LIN {X 0,Y 185.921,Z 403.304,A -85,B 0,C 180,E1 -22144.336,E2 -22144.336} C_VEL
LIN {X 0,Y 186.01,Z 403.316,A -85,B 0,C 180,E1 -22148.693,E2 -22148.693} C_VEL
LIN {X 0,Y 185.73,Z 403.33,A -85,B 0,C 180,E1 -22153.123,E2 -22153.123} C_VEL
LIN {X 0,Y 185.687,Z 403.347,A -85,B 0,C 180,E1 -22157.625,E2 -22157.625} C_VEL
LIN {X 0,Y 185.594,Z 403.365,A -85,B 0,C 180,E1 -22162.252,E2 -22162.252} C_VEL
LIN {X 0,Y 185.56,Z 403.358,A -85,B 0,C 180,E1 -22167.033,E2 -22167.033} C_VEL
LIN {X 0,Y 185.577,Z 403.368,A -85,B 0,C 180,E1 -22169.494,E2 -22169.494} C_VEL
LIN {X 0,Y 185.519,Z 403.376,A -85,B 0,C 180,E1 -22174.628,E2 -22174.628} C_VEL
LIN {X 0,Y 185.566,Z 403.36,A -85,B 0,C 180,E1 -22177.315,E2 -22177.315} C_VEL
LIN {X 0,Y 185.55,Z 403.372,A -85,B 0,C 180,E1 -22182.714,E2 -22182.714} C_VEL
LIN {X 0,Y 186.617,Z 406.323,A -85,B 0,C 180,E1 -22183.284,E2 -22183.284} C_VEL
LIN {X 0,Y 188.84,Z 408.797,A -85,B 0,C 180,E1 -22184.136,E2 -22184.136} C_VEL
LIN {X 0,Y 191.014,Z 412.188,A -85,B 0,C 180,E1 -22184.989,E2 -22184.989} C_VEL
LIN {X 0,Y 195.537,Z 418.863,A -85,B 0,C 180,E1 -22186.645,E2 -22186.645} C_VEL
LIN {X 0,Y 201.722,Z 428.495,A -85,B 0,C 180,E1 -22188.749,E2 -22188.749} C_VEL
LIN {X 0,Y 207.782,Z 439.318,A -85,B 0,C 180,E1 -22190.69,E2 -22190.69} C_VEL
LIN {X 0,Y 213.567,Z 452.7,A -85,B 0,C 180,E1 -22192.522,E2 -22192.522} C_VEL
LIN {X 0,Y 210.915,Z 504.609,A -85,B 0,C 180,E1 -22194.192,E2 -22194.192} C_VEL
LIN {X 0,Y 209.49,Z 518.077,A -85,B 0,C 180,E1 -22194.967,E2 -22194.967} C_VEL
LIN {X 0,Y 207.656,Z 530.461,A -85,B 0,C 180,E1 -22196.053,E2 -22196.053} C_VEL
LIN {X 0,Y 205.445,Z 541.745,A -85,B 0,C 180,E1 -22197.4,E2 -22197.4} C_VEL
LIN {X 0,Y 202.501,Z 553.363,A -85,B 0,C 180,E1 -22199.209,E2 -22199.209} C_VEL
LIN {X 0,Y 199.478,Z 563.795,A -85,B 0,C 180,E1 -22201.313,E2 -22201.313} C_VEL
LIN {X 0,Y 196.545,Z 573.207,A -85,B 0,C 180,E1 -22203.746,E2 -22203.746} C_VEL
LIN {X 0,Y 193.541,Z 581.541,A -85,B 0,C 180,E1 -22206.457,E2 -22206.457} C_VEL
LIN {X 0,Y 190.637,Z 588.935,A -85,B 0,C 180,E1 -22209.499,E2 -22209.499} C_VEL
LIN {X 0,Y 188.268,Z 594.864,A -85,B 0,C 180,E1 -22212.625,E2 -22212.625} C_VEL
LIN {X 0,Y 186.375,Z 599.545,A -85,B 0,C 180,E1 -22215.812,E2 -22215.812} C_VEL
LIN {X 0,Y 184.953,Z 603.125,A -85,B 0,C 180,E1 -22219.048,E2 -22219.048} C_VEL
LIN {X 0,Y 184.328,Z 604.97,A -85,B 0,C 180,E1 -22221.228,E2 -22221.228} C_VEL
LIN {X 0,Y 183.741,Z 606.644,A -85,B 0,C 180,E1 -22223.984,E2 -22223.984} C_VEL
LIN {X 0,Y 183.371,Z 607.945,A -85,B 0,C 180,E1 -22227.804,E2 -22227.804} C_VEL
LIN {X 0,Y 183.338,Z 608.171,A -85,B 0,C 180,E1 -22230,E2 -22230} C_VEL
LIN {X 0,Y 183.371,Z 607.978,A -85,B 0,C 180,E1 -22232.196,E2 -22232.196} C_VEL
LIN {X 0,Y 183.863,Z 606.429,A -85,B 0,C 180,E1 -22236.585,E2 -22236.585} C_VEL
LIN {X 0,Y 184.335,Z 605.076,A -85,B 0,C 180,E1 -22238.772,E2 -22238.772} C_VEL
LIN {X 0,Y 185.378,Z 602.216,A -85,B 0,C 180,E1 -22242.035,E2 -22242.035} C_VEL
LIN {X 0,Y 186.907,Z 598.332,A -85,B 0,C 180,E1 -22245.26,E2 -22245.26} C_VEL
LIN {X 0,Y 188.94,Z 593.319,A -85,B 0,C 180,E1 -22248.431,E2 -22248.431} C_VEL
LIN {X 0,Y 191.442,Z 587.001,A -85,B 0,C 180,E1 -22251.537,E2 -22251.537} C_VEL
LIN {X 0,Y 194.562,Z 579.089,A -85,B 0,C 180,E1 -22254.544,E2 -22254.544} C_VEL
LIN {X 0,Y 197.341,Z 570.784,A -85,B 0,C 180,E1 -22257.084,E2 -22257.084} C_VEL
LIN {X 0,Y 200.308,Z 561.19,A -85,B 0,C 180,E1 -22259.419,E2 -22259.419} C_VEL
LIN {X 0,Y 203.474,Z 550.096,A -85,B 0,C 180,E1 -22261.494,E2 -22261.494} C_VEL
LIN {X 0,Y 206.094,Z 539.217,A -85,B 0,C 180,E1 -22263.066,E2 -22263.066} C_VEL
LIN {X 0,Y 208.333,Z 527.192,A -85,B 0,C 180,E1 -22264.405,E2 -22264.405} C_VEL
LIN {X 0,Y 210.09,Z 514.712,A -85,B 0,C 180,E1 -22265.396,E2 -22265.396} C_VEL
LIN {X 0,Y 211.224,Z 502.268,A -85,B 0,C 180,E1 -22266.031,E2 -22266.031} C_VEL
LIN {X 0,Y 213.724,Z 452.937,A -85,B 0,C 180,E1 -22267.597,E2 -22267.597} C_VEL
LIN {X 0,Y 207.739,Z 439.055,A -85,B 0,C 180,E1 -22269.499,E2 -22269.499} C_VEL
LIN {X 0,Y 200.977,Z 427.208,A -85,B 0,C 180,E1 -22271.676,E2 -22271.676} C_VEL
LIN {X 0,Y 193.998,Z 416.477,A -85,B 0,C 180,E1 -22274.097,E2 -22274.097} C_VEL
LIN {X 0,Y 190.918,Z 412.068,A -85,B 0,C 180,E1 -22275.238,E2 -22275.238} C_VEL
LIN {X 0,Y 188.798,Z 408.673,A -85,B 0,C 180,E1 -22276.079,E2 -22276.079} C_VEL
LIN {X 0,Y 186.321,Z 405.856,A -85,B 0,C 180,E1 -22277.039,E2 -22277.039} C_VEL
LIN {X 0,Y 185.526,Z 403.347,A -85,B 0,C 180,E1 -22277.471,E2 -22277.471} C_VEL
LIN {X 0,Y 185.558,Z 403.363,A -85,B 0,C 180,E1 -22282.699,E2 -22282.699} C_VEL
LIN {X 0,Y 185.543,Z 403.368,A -85,B 0,C 180,E1 -22287.975,E2 -22287.975} C_VEL
LIN {X 0,Y 185.58,Z 403.361,A -85,B 0,C 180,E1 -22290.575,E2 -22290.575} C_VEL
LIN {X 0,Y 185.585,Z 403.361,A -85,B 0,C 180,E1 -22295.382,E2 -22295.382} C_VEL
LIN {X 0,Y 185.672,Z 403.349,A -85,B 0,C 180,E1 -22301.133,E2 -22301.133} C_VEL
LIN {X 0,Y 185.691,Z 403.351,A -85,B 0,C 180,E1 -22304.637,E2 -22304.637} C_VEL
LIN {X 0,Y 185.921,Z 403.311,A -85,B 0,C 180,E1 -22309.359,E2 -22309.359} C_VEL
LIN {X 0,Y 185.957,Z 403.316,A -85,B 0,C 180,E1 -22313.49,E2 -22313.49} C_VEL
LIN {X 0,Y 186.204,Z 403.289,A -85,B 0,C 180,E1 -22317.837,E2 -22317.837} C_VEL
LIN {X 0,Y 186.405,Z 403.263,A -85,B 0,C 180,E1 -22320,E2 -22320} C_VEL
LIN {X 0,Y 185.922,Z 403.322,A -85,B 0,C 180,E1 -22324.336,E2 -22324.336} C_VEL
LIN {X 0,Y 186.005,Z 403.299,A -85,B 0,C 180,E1 -22328.693,E2 -22328.693} C_VEL
LIN {X 0,Y 185.76,Z 403.336,A -85,B 0,C 180,E1 -22333.121,E2 -22333.121} C_VEL
LIN {X 0,Y 185.672,Z 403.347,A -85,B 0,C 180,E1 -22338.867,E2 -22338.867} C_VEL
LIN {X 0,Y 185.594,Z 403.367,A -85,B 0,C 180,E1 -22342.252,E2 -22342.252} C_VEL
LIN {X 0,Y 185.56,Z 403.371,A -85,B 0,C 180,E1 -22347.032,E2 -22347.032} C_VEL
LIN {X 0,Y 185.577,Z 403.367,A -85,B 0,C 180,E1 -22349.494,E2 -22349.494} C_VEL
LIN {X 0,Y 185.519,Z 403.368,A -85,B 0,C 180,E1 -22354.628,E2 -22354.628} C_VEL
LIN {X 0,Y 185.567,Z 403.437,A -85,B 0,C 180,E1 -22359.373,E2 -22359.373} C_VEL
LIN {X 0,Y 186.903,Z 408.111,A -85,B 0,C 180,E1 -22362.794,E2 -22362.794} C_VEL
LIN {X 0,Y 189.35,Z 412.41,A -85,B 0,C 180,E1 -22363.811,E2 -22363.811} C_VEL
LIN {X 0,Y 190.852,Z 414.784,A -85,B 0,C 180,E1 -22364.4,E2 -22364.4} C_VEL
LIN {X 0,Y 196.066,Z 423.736,A -85,B 0,C 180,E1 -22366.366,E2 -22366.366} C_VEL
LIN {X 0,Y 202.742,Z 436.785,A -85,B 0,C 180,E1 -22368.727,E2 -22368.727} C_VEL
LIN {X 0,Y 209.741,Z 452.959,A -85,B 0,C 180,E1 -22371.069,E2 -22371.069} C_VEL
LIN {X 0,Y 211.194,Z 456.662,A -85,B 0,C 180,E1 -22371.542,E2 -22371.542} C_VEL
LIN {X 0,Y 212.839,Z 470.861,A -85,B 0,C 180,E1 -22372.482,E2 -22372.482} C_VEL
LIN {X 0,Y 211.219,Z 504.612,A -85,B 0,C 180,E1 -22373.552,E2 -22373.552} C_VEL
LIN {X 0,Y 210.385,Z 510.464,A -85,B 0,C 180,E1 -22373.628,E2 -22373.628} C_VEL
LIN {X 0,Y 207.304,Z 519.917,A -85,B 0,C 180,E1 -22373.522,E2 -22373.522} C_VEL
LIN {X 0,Y 203.883,Z 529.234,A -85,B 0,C 180,E1 -22373.577,E2 -22373.577} C_VEL
LIN {X 0,Y 202.499,Z 534.867,A -85,B 0,C 180,E1 -22373.897,E2 -22373.897} C_VEL
LIN {X 0,Y 199.9,Z 547.969,A -85,B 0,C 180,E1 -22375.159,E2 -22375.159} C_VEL
LIN {X 0,Y 196.981,Z 559.755,A -85,B 0,C 180,E1 -22376.733,E2 -22376.733} C_VEL
LIN {X 0,Y 193.867,Z 570.352,A -85,B 0,C 180,E1 -22378.594,E2 -22378.594} C_VEL
LIN {X 0,Y 190.595,Z 580.039,A -85,B 0,C 180,E1 -22380.753,E2 -22380.753} C_VEL
LIN {X 0,Y 187.348,Z 588.873,A -85,B 0,C 180,E1 -22383.247,E2 -22383.247} C_VEL
LIN {X 0,Y 184.148,Z 597.424,A -85,B 0,C 180,E1 -22386.343,E2 -22386.343} C_VEL
LIN {X 0,Y 181.905,Z 603.374,A -85,B 0,C 180,E1 -22389.061,E2 -22389.061} C_VEL
LIN {X 0,Y 179.971,Z 608.236,A -85,B 0,C 180,E1 -22391.796,E2 -22391.796} C_VEL
LIN {X 0,Y 178.081,Z 612.962,A -85,B 0,C 180,E1 -22395.136,E2 -22395.136} C_VEL
LIN {X 0,Y 176.948,Z 616.585,A -85,B 0,C 180,E1 -22398.546,E2 -22398.546} C_VEL
LIN {X 0,Y 176.45,Z 618.455,A -85,B 0,C 180,E1 -22400.833,E2 -22400.833} C_VEL
LIN {X 0,Y 176.137,Z 619.86,A -85,B 0,C 180,E1 -22403.125,E2 -22403.125} C_VEL
LIN {X 0,Y 175.991,Z 621.264,A -85,B 0,C 180,E1 -22406.709,E2 -22406.709} C_VEL
LIN {X 0,Y 176.185,Z 621.701,A -85,B 0,C 180,E1 -22410,E2 -22410} C_VEL
LIN {X 0,Y 175.996,Z 621.246,A -85,B 0,C 180,E1 -22413.32,E2 -22413.32} C_VEL
LIN {X 0,Y 176.135,Z 619.831,A -85,B 0,C 180,E1 -22416.875,E2 -22416.875} C_VEL
LIN {X 0,Y 176.444,Z 618.412,A -85,B 0,C 180,E1 -22419.168,E2 -22419.168} C_VEL
LIN {X 0,Y 177.285,Z 615.445,A -85,B 0,C 180,E1 -22422.593,E2 -22422.593} C_VEL
LIN {X 0,Y 178.607,Z 611.438,A -85,B 0,C 180,E1 -22425.988,E2 -22425.988} C_VEL
LIN {X 0,Y 181.065,Z 605.294,A -85,B 0,C 180,E1 -22429.854,E2 -22429.854} C_VEL
LIN {X 0,Y 184.117,Z 597.764,A -85,B 0,C 180,E1 -22433.431,E2 -22433.431} C_VEL
LIN {X 0,Y 186.819,Z 590.279,A -85,B 0,C 180,E1 -22436.233,E2 -22436.233} C_VEL
LIN {X 0,Y 189.965,Z 581.763,A -85,B 0,C 180,E1 -22438.747,E2 -22438.747} C_VEL
LIN {X 0,Y 193.48,Z 571.246,A -85,B 0,C 180,E1 -22441.172,E2 -22441.172} C_VEL
LIN {X 0,Y 196.972,Z 559.412,A -85,B 0,C 180,E1 -22443.269,E2 -22443.269} C_VEL
LIN {X 0,Y 199.884,Z 547.485,A -85,B 0,C 180,E1 -22444.844,E2 -22444.844} C_VEL
LIN {X 0,Y 202.319,Z 535.072,A -85,B 0,C 180,E1 -22446.04,E2 -22446.04} C_VEL
LIN {X 0,Y 204.168,Z 522.069,A -85,B 0,C 180,E1 -22446.901,E2 -22446.901} C_VEL
LIN {X 0,Y 205.296,Z 506.698,A -85,B 0,C 180,E1 -22447.502,E2 -22447.502} C_VEL
LIN {X 0,Y 207.019,Z 471.198,A -85,B 0,C 180,E1 -22448.664,E2 -22448.664} C_VEL
LIN {X 0,Y 205.496,Z 458.664,A -85,B 0,C 180,E1 -22449.553,E2 -22449.553} C_VEL
LIN {X 0,Y 198.861,Z 442.643,A -85,B 0,C 180,E1 -22451.888,E2 -22451.888} C_VEL
LIN {X 0,Y 192.918,Z 430.579,A -85,B 0,C 180,E1 -22454.081,E2 -22454.081} C_VEL
LIN {X 0,Y 188.154,Z 422.026,A -85,B 0,C 180,E1 -22455.944,E2 -22455.944} C_VEL
LIN {X 0,Y 185.548,Z 417.623,A -85,B 0,C 180,E1 -22457.017,E2 -22457.017} C_VEL
LIN {X 0,Y 182.438,Z 412.577,A -85,B 0,C 180,E1 -22458.355,E2 -22458.355} C_VEL
LIN {X 0,Y 179.779,Z 408.407,A -85,B 0,C 180,E1 -22459.557,E2 -22459.557} C_VEL
LIN {X 0,Y 179.458,Z 407.656,A -85,B 0,C 180,E1 -22459.746,E2 -22459.746} C_VEL
LIN {X 0,Y 178.528,Z 404.239,A -85,B 0,C 180,E1 -22462.488,E2 -22462.488} C_VEL
LIN {X 0,Y 178.489,Z 404.24,A -85,B 0,C 180,E1 -22466.547,E2 -22466.547} C_VEL
LIN {X 0,Y 178.52,Z 404.239,A -85,B 0,C 180,E1 -22470.006,E2 -22470.006} C_VEL
LIN {X 0,Y 178.532,Z 404.238,A -85,B 0,C 180,E1 -22474.875,E2 -22474.875} C_VEL
LIN {X 0,Y 178.62,Z 404.229,A -85,B 0,C 180,E1 -22480.784,E2 -22480.784} C_VEL
LIN {X 0,Y 178.657,Z 404.231,A -85,B 0,C 180,E1 -22486.348,E2 -22486.348} C_VEL
LIN {X 0,Y 178.934,Z 404.179,A -85,B 0,C 180,E1 -22490.961,E2 -22490.961} C_VEL
LIN {X 0,Y 179.149,Z 404.148,A -85,B 0,C 180,E1 -22497.752,E2 -22497.752} C_VEL
LIN {X 0,Y 179.368,Z 404.14,A -85,B 0,C 180,E1 -22500,E2 -22500} C_VEL
LIN {X 0,Y 178.869,Z 404.181,A -85,B 0,C 180,E1 -22504.507,E2 -22504.507} C_VEL
LIN {X 0,Y 178.96,Z 404.192,A -85,B 0,C 180,E1 -22509.038,E2 -22509.038} C_VEL
LIN {X 0,Y 178.657,Z 404.214,A -85,B 0,C 180,E1 -22513.652,E2 -22513.652} C_VEL
LIN {X 0,Y 178.62,Z 404.215,A -85,B 0,C 180,E1 -22519.216,E2 -22519.216} C_VEL
LIN {X 0,Y 178.522,Z 404.232,A -85,B 0,C 180,E1 -22525.118,E2 -22525.118} C_VEL
LIN {X 0,Y 178.521,Z 404.242,A -85,B 0,C 180,E1 -22529.994,E2 -22529.994} C_VEL
LIN {X 0,Y 178.483,Z 404.253,A -85,B 0,C 180,E1 -22534.22,E2 -22534.22} C_VEL
LIN {X 0,Y 178.477,Z 404.249,A -85,B 0,C 180,E1 -22539.784,E2 -22539.784} C_VEL
LIN {X 0,Y 178.499,Z 404.253,A -85,B 0,C 180,E1 -22540.284,E2 -22540.284} C_VEL
LIN {X 0,Y 179.432,Z 406.939,A -85,B 0,C 180,E1 -22540.8,E2 -22540.8} C_VEL
LIN {X 0,Y 181.274,Z 409.049,A -85,B 0,C 180,E1 -22541.601,E2 -22541.601} C_VEL
LIN {X 0,Y 181.942,Z 409.687,A -85,B 0,C 180,E1 -22541.877,E2 -22541.877} C_VEL
LIN {X 0,Y 184.131,Z 413.133,A -85,B 0,C 180,E1 -22542.834,E2 -22542.834} C_VEL
LIN {X 0,Y 185.375,Z 414.712,A -85,B 0,C 180,E1 -22543.339,E2 -22543.339} C_VEL
LIN {X 0,Y 193.39,Z 426.657,A -85,B 0,C 180,E1 -22546.43,E2 -22546.43} C_VEL
LIN {X 0,Y 200.319,Z 438.22,A -85,B 0,C 180,E1 -22548.849,E2 -22548.849} C_VEL
LIN {X 0,Y 204.76,Z 447.222,A -85,B 0,C 180,E1 -22550.342,E2 -22550.342} C_VEL
LIN {X 0,Y 207.962,Z 454.895,A -85,B 0,C 180,E1 -22551.411,E2 -22551.411} C_VEL
LIN {X 0,Y 205.194,Z 505.053,A -85,B 0,C 180,E1 -22553.041,E2 -22553.041} C_VEL
LIN {X 0,Y 203.704,Z 518.479,A -85,B 0,C 180,E1 -22553.83,E2 -22553.83} C_VEL
LIN {X 0,Y 201.823,Z 530.735,A -85,B 0,C 180,E1 -22554.931,E2 -22554.931} C_VEL
LIN {X 0,Y 199.521,Z 542.016,A -85,B 0,C 180,E1 -22556.305,E2 -22556.305} C_VEL
LIN {X 0,Y 196.448,Z 553.634,A -85,B 0,C 180,E1 -22558.152,E2 -22558.152} C_VEL
LIN {X 0,Y 193.271,Z 564.066,A -85,B 0,C 180,E1 -22560.301,E2 -22560.301} C_VEL
LIN {X 0,Y 190.101,Z 573.75,A -85,B 0,C 180,E1 -22562.883,E2 -22562.883} C_VEL
LIN {X 0,Y 187.061,Z 581.81,A -85,B 0,C 180,E1 -22565.59,E2 -22565.59} C_VEL
LIN {X 0,Y 184.018,Z 589.204,A -85,B 0,C 180,E1 -22568.727,E2 -22568.727} C_VEL
LIN {X 0,Y 181.519,Z 595.132,A -85,B 0,C 180,E1 -22571.957,E2 -22571.957} C_VEL
LIN {X 0,Y 179.504,Z 599.814,A -85,B 0,C 180,E1 -22575.257,E2 -22575.257} C_VEL
LIN {X 0,Y 178.004,Z 603.393,A -85,B 0,C 180,E1 -22578.615,E2 -22578.615} C_VEL
LIN {X 0,Y 177.309,Z 605.238,A -85,B 0,C 180,E1 -22580.878,E2 -22580.878} C_VEL
LIN {X 0,Y 176.658,Z 607.052,A -85,B 0,C 180,E1 -22584.034,E2 -22584.034} C_VEL
LIN {X 0,Y 176.281,Z 608.213,A -85,B 0,C 180,E1 -22587.715,E2 -22587.715} C_VEL
LIN {X 0,Y 176.243,Z 608.438,A -85,B 0,C 180,E1 -22590,E2 -22590} C_VEL
LIN {X 0,Y 176.281,Z 608.245,A -85,B 0,C 180,E1 -22592.285,E2 -22592.285} C_VEL
LIN {X 0,Y 176.816,Z 606.696,A -85,B 0,C 180,E1 -22596.848,E2 -22596.848} C_VEL
LIN {X 0,Y 177.315,Z 605.343,A -85,B 0,C 180,E1 -22599.122,E2 -22599.122} C_VEL
LIN {X 0,Y 178.454,Z 602.481,A -85,B 0,C 180,E1 -22602.509,E2 -22602.509} C_VEL
LIN {X 0,Y 180.072,Z 598.598,A -85,B 0,C 180,E1 -22605.854,E2 -22605.854} C_VEL
LIN {X 0,Y 182.209,Z 593.585,A -85,B 0,C 180,E1 -22609.138,E2 -22609.138} C_VEL
LIN {X 0,Y 184.877,Z 587.266,A -85,B 0,C 180,E1 -22612.342,E2 -22612.342} C_VEL
LIN {X 0,Y 188.143,Z 579.353,A -85,B 0,C 180,E1 -22615.44,E2 -22615.44} C_VEL
LIN {X 0,Y 191.21,Z 570.575,A -85,B 0,C 180,E1 -22618.187,E2 -22618.187} C_VEL
LIN {X 0,Y 194.524,Z 560.352,A -85,B 0,C 180,E1 -22620.685,E2 -22620.685} C_VEL
LIN {X 0,Y 197.833,Z 548.937,A -85,B 0,C 180,E1 -22622.802,E2 -22622.802} C_VEL
LIN {X 0,Y 200.611,Z 537.717,A -85,B 0,C 180,E1 -22624.395,E2 -22624.395} C_VEL
LIN {X 0,Y 202.732,Z 526.313,A -85,B 0,C 180,E1 -22625.649,E2 -22625.649} C_VEL
LIN {X 0,Y 204.541,Z 513.346,A -85,B 0,C 180,E1 -22626.645,E2 -22626.645} C_VEL
LIN {X 0,Y 205.564,Z 501.19,A -85,B 0,C 180,E1 -22627.256,E2 -22627.256} C_VEL
LIN {X 0,Y 208.012,Z 454.901,A -85,B 0,C 180,E1 -22628.744,E2 -22628.744} C_VEL
LIN {X 0,Y 202.668,Z 442.523,A -85,B 0,C 180,E1 -22630.543,E2 -22630.543} C_VEL
LIN {X 0,Y 196.607,Z 431.784,A -85,B 0,C 180,E1 -22632.607,E2 -22632.607} C_VEL
LIN {X 0,Y 189.994,Z 421.47,A -85,B 0,C 180,E1 -22635.025,E2 -22635.025} C_VEL
LIN {X 0,Y 186.453,Z 416.413,A -85,B 0,C 180,E1 -22636.412,E2 -22636.412} C_VEL
LIN {X 0,Y 184.428,Z 413.419,A -85,B 0,C 180,E1 -22637.251,E2 -22637.251} C_VEL
LIN {X 0,Y 182.216,Z 410.251,A -85,B 0,C 180,E1 -22638.2,E2 -22638.2} C_VEL
LIN {X 0,Y 181.444,Z 409.171,A -85,B 0,C 180,E1 -22638.539,E2 -22638.539} C_VEL
LIN {X 0,Y 179.347,Z 406.852,A -85,B 0,C 180,E1 -22639.45,E2 -22639.45} C_VEL
LIN {X 0,Y 178.501,Z 404.246,A -85,B 0,C 180,E1 -22639.947,E2 -22639.947} C_VEL
LIN {X 0,Y 178.457,Z 404.252,A -85,B 0,C 180,E1 -22643.791,E2 -22643.791} C_VEL
LIN {X 0,Y 178.489,Z 404.242,A -85,B 0,C 180,E1 -22646.547,E2 -22646.547} C_VEL
LIN {X 0,Y 178.521,Z 404.244,A -85,B 0,C 180,E1 -22650.006,E2 -22650.006} C_VEL
LIN {X 0,Y 178.532,Z 404.244,A -85,B 0,C 180,E1 -22654.875,E2 -22654.875} C_VEL
LIN {X 0,Y 178.62,Z 404.23,A -85,B 0,C 180,E1 -22660.784,E2 -22660.784} C_VEL
LIN {X 0,Y 178.657,Z 404.23,A -85,B 0,C 180,E1 -22666.348,E2 -22666.348} C_VEL
LIN {X 0,Y 178.956,Z 404.189,A -85,B 0,C 180,E1 -22670.962,E2 -22670.962} C_VEL
LIN {X 0,Y 179.149,Z 404.166,A -85,B 0,C 180,E1 -22677.752,E2 -22677.752} C_VEL
LIN {X 0,Y 179.368,Z 404.138,A -85,B 0,C 180,E1 -22680,E2 -22680} C_VEL
LIN {X 0,Y 178.87,Z 404.201,A -85,B 0,C 180,E1 -22684.507,E2 -22684.507} C_VEL
LIN {X 0,Y 178.934,Z 404.18,A -85,B 0,C 180,E1 -22689.039,E2 -22689.039} C_VEL
LIN {X 0,Y 178.678,Z 404.215,A -85,B 0,C 180,E1 -22693.651,E2 -22693.651} C_VEL
LIN {X 0,Y 178.62,Z 404.223,A -85,B 0,C 180,E1 -22699.216,E2 -22699.216} C_VEL
LIN {X 0,Y 178.522,Z 404.238,A -85,B 0,C 180,E1 -22705.118,E2 -22705.118} C_VEL
LIN {X 0,Y 178.52,Z 404.245,A -85,B 0,C 180,E1 -22709.994,E2 -22709.994} C_VEL
LIN {X 0,Y 178.483,Z 404.241,A -85,B 0,C 180,E1 -22714.22,E2 -22714.22} C_VEL
LIN {X 0,Y 178.544,Z 404.366,A -85,B 0,C 180,E1 -22717.515,E2 -22717.515} C_VEL
LIN {X 0,Y 179.463,Z 407.711,A -85,B 0,C 180,E1 -22720.161,E2 -22720.161} C_VEL
LIN {X 0,Y 182.34,Z 412.457,A -85,B 0,C 180,E1 -22721.488,E2 -22721.488} C_VEL
LIN {X 0,Y 184.139,Z 415.339,A -85,B 0,C 180,E1 -22722.275,E2 -22722.275} C_VEL
LIN {X 0,Y 186.975,Z 419.928,A -85,B 0,C 180,E1 -22723.465,E2 -22723.465} C_VEL
LIN {X 0,Y 192.107,Z 429.035,A -85,B 0,C 180,E1 -22725.511,E2 -22725.511} C_VEL
LIN {X 0,Y 197.957,Z 440.605,A -85,B 0,C 180,E1 -22727.694,E2 -22727.694} C_VEL
LIN {X 0,Y 204.803,Z 456.726,A -85,B 0,C 180,E1 -22730.123,E2 -22730.123} C_VEL
LIN {X 0,Y 205.871,Z 459.872,A -85,B 0,C 180,E1 -22730.507,E2 -22730.507} C_VEL
LIN {X 0,Y 207.17,Z 472.203,A -85,B 0,C 180,E1 -22731.337,E2 -22731.337} C_VEL
LIN {X 0,Y 204.731,Z 518.229,A -85,B 0,C 180,E1 -22732.882,E2 -22732.882} C_VEL
LIN {X 0,Y 203.028,Z 531.674,A -85,B 0,C 180,E1 -22733.656,E2 -22733.656} C_VEL
LIN {X 0,Y 202.499,Z 534.867,A -85,B 0,C 180,E1 -22733.897,E2 -22733.897} C_VEL
LIN {X 0,Y 200.968,Z 540.521,A -85,B 0,C 180,E1 -22734.284,E2 -22734.284} C_VEL
LIN {X 0,Y 196.735,Z 549.398,A -85,B 0,C 180,E1 -22734.769,E2 -22734.769} C_VEL
LIN {X 0,Y 192.146,Z 557.81,A -85,B 0,C 180,E1 -22735.426,E2 -22735.426} C_VEL
LIN {X 0,Y 190.103,Z 562.779,A -85,B 0,C 180,E1 -22736.1,E2 -22736.1} C_VEL
LIN {X 0,Y 186.67,Z 573.565,A -85,B 0,C 180,E1 -22738.192,E2 -22738.192} C_VEL
LIN {X 0,Y 183.027,Z 583.515,A -85,B 0,C 180,E1 -22740.688,E2 -22740.688} C_VEL
LIN {X 0,Y 179.796,Z 591.68,A -85,B 0,C 180,E1 -22743.288,E2 -22743.288} C_VEL
LIN {X 0,Y 176.715,Z 599.71,A -85,B 0,C 180,E1 -22746.566,E2 -22746.566} C_VEL
LIN {X 0,Y 173.989,Z 606.143,A -85,B 0,C 180,E1 -22749.92,E2 -22749.92} C_VEL
LIN {X 0,Y 171.777,Z 611.256,A -85,B 0,C 180,E1 -22753.358,E2 -22753.358} C_VEL
LIN {X 0,Y 170.313,Z 615.238,A -85,B 0,C 180,E1 -22756.882,E2 -22756.882} C_VEL
LIN {X 0,Y 169.406,Z 618.187,A -85,B 0,C 180,E1 -22760.448,E2 -22760.448} C_VEL
LIN {X 0,Y 169.071,Z 619.592,A -85,B 0,C 180,E1 -22762.836,E2 -22762.836} C_VEL
LIN {X 0,Y 168.899,Z 621.092,A -85,B 0,C 180,E1 -22767.028,E2 -22767.028} C_VEL
LIN {X 0,Y 169.089,Z 621.434,A -85,B 0,C 180,E1 -22770,E2 -22770} C_VEL
LIN {X 0,Y 168.93,Z 621.04,A -85,B 0,C 180,E1 -22773.163,E2 -22773.163} C_VEL
LIN {X 0,Y 169.068,Z 619.562,A -85,B 0,C 180,E1 -22777.164,E2 -22777.164} C_VEL
LIN {X 0,Y 169.401,Z 618.143,A -85,B 0,C 180,E1 -22779.552,E2 -22779.552} C_VEL
LIN {X 0,Y 170.311,Z 615.175,A -85,B 0,C 180,E1 -22783.118,E2 -22783.118} C_VEL
LIN {X 0,Y 171.774,Z 611.169,A -85,B 0,C 180,E1 -22786.642,E2 -22786.642} C_VEL
LIN {X 0,Y 174.355,Z 605.024,A -85,B 0,C 180,E1 -22790.652,E2 -22790.652} C_VEL
LIN {X 0,Y 177.339,Z 598.098,A -85,B 0,C 180,E1 -22794.079,E2 -22794.079} C_VEL
LIN {X 0,Y 180.452,Z 590.008,A -85,B 0,C 180,E1 -22797.233,E2 -22797.233} C_VEL
LIN {X 0,Y 183.76,Z 581.492,A -85,B 0,C 180,E1 -22799.814,E2 -22799.814} C_VEL
LIN {X 0,Y 187.445,Z 570.976,A -85,B 0,C 180,E1 -22802.294,E2 -22802.294} C_VEL
LIN {X 0,Y 190.655,Z 560.572,A -85,B 0,C 180,E1 -22804.204,E2 -22804.204} C_VEL
LIN {X 0,Y 193.66,Z 549.159,A -85,B 0,C 180,E1 -22805.815,E2 -22805.815} C_VEL
LIN {X 0,Y 196.154,Z 537.4,A -85,B 0,C 180,E1 -22807.039,E2 -22807.039} C_VEL
LIN {X 0,Y 198.273,Z 523.822,A -85,B 0,C 180,E1 -22808.016,E2 -22808.016} C_VEL
LIN {X 0,Y 199.49,Z 510.457,A -85,B 0,C 180,E1 -22808.611,E2 -22808.611} C_VEL
LIN {X 0,Y 201.467,Z 472.332,A -85,B 0,C 180,E1 -22809.874,E2 -22809.874} C_VEL
LIN {X 0,Y 200.186,Z 461.38,A -85,B 0,C 180,E1 -22810.682,E2 -22810.682} C_VEL
LIN {X 0,Y 193.754,Z 445.675,A -85,B 0,C 180,E1 -22813.093,E2 -22813.093} C_VEL
LIN {X 0,Y 187.871,Z 433.538,A -85,B 0,C 180,E1 -22815.418,E2 -22815.418} C_VEL
LIN {X 0,Y 181.729,Z 422.646,A -85,B 0,C 180,E1 -22818.022,E2 -22818.022} C_VEL
LIN {X 0,Y 178.684,Z 417.711,A -85,B 0,C 180,E1 -22819.403,E2 -22819.403} C_VEL
LIN {X 0,Y 175.209,Z 412.284,A -85,B 0,C 180,E1 -22821.077,E2 -22821.077} C_VEL
LIN {X 0,Y 172.553,Z 408.312,A -85,B 0,C 180,E1 -22822.434,E2 -22822.434} C_VEL
LIN {X 0,Y 172.071,Z 407.183,A -85,B 0,C 180,E1 -22822.771,E2 -22822.771} C_VEL
LIN {X 0,Y 171.426,Z 405.132,A -85,B 0,C 180,E1 -22824.794,E2 -22824.794} C_VEL
LIN {X 0,Y 171.456,Z 405.124,A -85,B 0,C 180,E1 -22829.404,E2 -22829.404} C_VEL
LIN {X 0,Y 171.467,Z 405.123,A -85,B 0,C 180,E1 -22834.383,E2 -22834.383} C_VEL
LIN {X 0,Y 171.576,Z 405.105,A -85,B 0,C 180,E1 -22840.871,E2 -22840.871} C_VEL
LIN {X 0,Y 171.574,Z 405.113,A -85,B 0,C 180,E1 -22845.773,E2 -22845.773} C_VEL
LIN {X 0,Y 171.869,Z 405.056,A -85,B 0,C 180,E1 -22850.586,E2 -22850.586} C_VEL
LIN {X 0,Y 171.817,Z 405.07,A -85,B 0,C 180,E1 -22855.308,E2 -22855.308} C_VEL
LIN {X 0,Y 172.331,Z 405.017,A -85,B 0,C 180,E1 -22860,E2 -22860} C_VEL
LIN {X 0,Y 171.818,Z 405.059,A -85,B 0,C 180,E1 -22864.693,E2 -22864.693} C_VEL
LIN {X 0,Y 171.887,Z 405.072,A -85,B 0,C 180,E1 -22869.413,E2 -22869.413} C_VEL
LIN {X 0,Y 171.574,Z 405.102,A -85,B 0,C 180,E1 -22874.228,E2 -22874.228} C_VEL
LIN {X 0,Y 171.541,Z 405.096,A -85,B 0,C 180,E1 -22879.562,E2 -22879.562} C_VEL
LIN {X 0,Y 171.46,Z 405.109,A -85,B 0,C 180,E1 -22885.612,E2 -22885.612} C_VEL
LIN {X 0,Y 171.439,Z 405.119,A -85,B 0,C 180,E1 -22890.587,E2 -22890.587} C_VEL
LIN {X 0,Y 171.433,Z 405.119,A -85,B 0,C 180,E1 -22896.473,E2 -22896.473} C_VEL
LIN {X 0,Y 171.42,Z 405.121,A -85,B 0,C 180,E1 -22897.394,E2 -22897.394} C_VEL
LIN {X 0,Y 172.504,Z 408.032,A -85,B 0,C 180,E1 -22898.101,E2 -22898.101} C_VEL
LIN {X 0,Y 174.511,Z 410.147,A -85,B 0,C 180,E1 -22899.078,E2 -22899.078} C_VEL
LIN {X 0,Y 175.23,Z 410.924,A -85,B 0,C 180,E1 -22899.419,E2 -22899.419} C_VEL
LIN {X 0,Y 177.341,Z 414.18,A -85,B 0,C 180,E1 -22900.451,E2 -22900.451} C_VEL
LIN {X 0,Y 178.765,Z 415.871,A -85,B 0,C 180,E1 -22901.09,E2 -22901.09} C_VEL
LIN {X 0,Y 182.731,Z 421.675,A -85,B 0,C 180,E1 -22902.842,E2 -22902.842} C_VEL
LIN {X 0,Y 189.016,Z 431.038,A -85,B 0,C 180,E1 -22905.373,E2 -22905.373} C_VEL
LIN {X 0,Y 195.768,Z 442.518,A -85,B 0,C 180,E1 -22907.872,E2 -22907.872} C_VEL
LIN {X 0,Y 200.089,Z 451.464,A -85,B 0,C 180,E1 -22909.41,E2 -22909.41} C_VEL
LIN {X 0,Y 202.342,Z 456.987,A -85,B 0,C 180,E1 -22910.211,E2 -22910.211} C_VEL
LIN {X 0,Y 199.529,Z 505.635,A -85,B 0,C 180,E1 -22911.828,E2 -22911.828} C_VEL
LIN {X 0,Y 198.009,Z 518.889,A -85,B 0,C 180,E1 -22912.63,E2 -22912.63} C_VEL
LIN {X 0,Y 196.065,Z 531.009,A -85,B 0,C 180,E1 -22913.741,E2 -22913.741} C_VEL
LIN {X 0,Y 193.669,Z 542.288,A -85,B 0,C 180,E1 -22915.143,E2 -22915.143} C_VEL
LIN {X 0,Y 190.466,Z 553.905,A -85,B 0,C 180,E1 -22917.027,E2 -22917.027} C_VEL
LIN {X 0,Y 187.134,Z 564.337,A -85,B 0,C 180,E1 -22919.224,E2 -22919.224} C_VEL
LIN {X 0,Y 184.207,Z 572.891,A -85,B 0,C 180,E1 -22921.531,E2 -22921.531} C_VEL
LIN {X 0,Y 181.213,Z 580.697,A -85,B 0,C 180,E1 -22924.132,E2 -22924.132} C_VEL
LIN {X 0,Y 177.887,Z 588.365,A -85,B 0,C 180,E1 -22927.344,E2 -22927.344} C_VEL
LIN {X 0,Y 174.774,Z 595.401,A -85,B 0,C 180,E1 -22931.235,E2 -22931.235} C_VEL
LIN {X 0,Y 172.659,Z 600.082,A -85,B 0,C 180,E1 -22934.658,E2 -22934.658} C_VEL
LIN {X 0,Y 171.053,Z 603.66,A -85,B 0,C 180,E1 -22938.145,E2 -22938.145} C_VEL
LIN {X 0,Y 170.292,Z 605.506,A -85,B 0,C 180,E1 -22940.498,E2 -22940.498} C_VEL
LIN {X 0,Y 169.505,Z 607.564,A -85,B 0,C 180,E1 -22944.32,E2 -22944.32} C_VEL
LIN {X 0,Y 169.194,Z 608.48,A -85,B 0,C 180,E1 -22947.619,E2 -22947.619} C_VEL
LIN {X 0,Y 169.151,Z 608.705,A -85,B 0,C 180,E1 -22950,E2 -22950} C_VEL
LIN {X 0,Y 169.194,Z 608.511,A -85,B 0,C 180,E1 -22952.381,E2 -22952.381} C_VEL
LIN {X 0,Y 169.783,Z 606.962,A -85,B 0,C 180,E1 -22957.133,E2 -22957.133} C_VEL
LIN {X 0,Y 170.298,Z 605.61,A -85,B 0,C 180,E1 -22959.501,E2 -22959.501} C_VEL
LIN {X 0,Y 171.525,Z 602.748,A -85,B 0,C 180,E1 -22963.023,E2 -22963.023} C_VEL
LIN {X 0,Y 173.263,Z 598.864,A -85,B 0,C 180,E1 -22966.495,E2 -22966.495} C_VEL
LIN {X 0,Y 175.513,Z 593.851,A -85,B 0,C 180,E1 -22969.898,E2 -22969.898} C_VEL
LIN {X 0,Y 178.337,Z 587.531,A -85,B 0,C 180,E1 -22973.208,E2 -22973.208} C_VEL
LIN {X 0,Y 181.767,Z 579.617,A -85,B 0,C 180,E1 -22976.4,E2 -22976.4} C_VEL
LIN {X 0,Y 184.887,Z 571.093,A -85,B 0,C 180,E1 -22979.153,E2 -22979.153} C_VEL
LIN {X 0,Y 188.094,Z 561.716,A -85,B 0,C 180,E1 -22981.54,E2 -22981.54} C_VEL
LIN {X 0,Y 191.544,Z 550.619,A -85,B 0,C 180,E1 -22983.707,E2 -22983.707} C_VEL
LIN {X 0,Y 194.385,Z 539.738,A -85,B 0,C 180,E1 -22985.343,E2 -22985.343} C_VEL
LIN {X 0,Y 196.819,Z 527.71,A -85,B 0,C 180,E1 -22986.733,E2 -22986.733} C_VEL
LIN {X 0,Y 198.694,Z 515.395,A -85,B 0,C 180,E1 -22987.751,E2 -22987.751} C_VEL
LIN {X 0,Y 199.952,Z 501.977,A -85,B 0,C 180,E1 -22988.46,E2 -22988.46} C_VEL
LIN {X 0,Y 202.429,Z 457.041,A -85,B 0,C 180,E1 -22989.938,E2 -22989.938} C_VEL
LIN {X 0,Y 197.576,Z 445.864,A -85,B 0,C 180,E1 -22991.669,E2 -22991.669} C_VEL
LIN {X 0,Y 190.944,Z 434.057,A -85,B 0,C 180,E1 -22994.087,E2 -22994.087} C_VEL
LIN {X 0,Y 183.585,Z 422.785,A -85,B 0,C 180,E1 -22997.008,E2 -22997.008} C_VEL
LIN {X 0,Y 180.713,Z 418.712,A -85,B 0,C 180,E1 -22998.241,E2 -22998.241} C_VEL
LIN {X 0,Y 177.941,Z 414.782,A -85,B 0,C 180,E1 -22999.499,E2 -22999.499} C_VEL
LIN {X 0,Y 175.597,Z 411.667,A -85,B 0,C 180,E1 -23000.608,E2 -23000.608} C_VEL
LIN {X 0,Y 174.824,Z 410.346,A -85,B 0,C 180,E1 -23001.005,E2 -23001.005} C_VEL
LIN {X 0,Y 172.683,Z 408.34,A -85,B 0,C 180,E1 -23002.032,E2 -23002.032} C_VEL
LIN {X 0,Y 171.603,Z 406.109,A -85,B 0,C 180,E1 -23002.652,E2 -23002.652} C_VEL
LIN {X 0,Y 171.407,Z 405.125,A -85,B 0,C 180,E1 -23002.833,E2 -23002.833} C_VEL
LIN {X 0,Y 171.426,Z 405.124,A -85,B 0,C 180,E1 -23007.794,E2 -23007.794} C_VEL
LIN {X 0,Y 171.447,Z 405.12,A -85,B 0,C 180,E1 -23010.534,E2 -23010.534} C_VEL
LIN {X 0,Y 171.455,Z 405.117,A -85,B 0,C 180,E1 -23015.801,E2 -23015.801} C_VEL
LIN {X 0,Y 171.576,Z 405.106,A -85,B 0,C 180,E1 -23020.871,E2 -23020.871} C_VEL
LIN {X 0,Y 171.575,Z 405.113,A -85,B 0,C 180,E1 -23025.772,E2 -23025.772} C_VEL
LIN {X 0,Y 171.885,Z 405.066,A -85,B 0,C 180,E1 -23030.587,E2 -23030.587} C_VEL
LIN {X 0,Y 171.817,Z 405.065,A -85,B 0,C 180,E1 -23035.307,E2 -23035.307} C_VEL
LIN {X 0,Y 172.331,Z 405.014,A -85,B 0,C 180,E1 -23040,E2 -23040} C_VEL
LIN {X 0,Y 171.819,Z 405.08,A -85,B 0,C 180,E1 -23044.692,E2 -23044.692} C_VEL
LIN {X 0,Y 171.87,Z 405.062,A -85,B 0,C 180,E1 -23049.414,E2 -23049.414} C_VEL
LIN {X 0,Y 171.59,Z 405.095,A -85,B 0,C 180,E1 -23054.226,E2 -23054.226} C_VEL
LIN {X 0,Y 171.541,Z 405.104,A -85,B 0,C 180,E1 -23059.562,E2 -23059.562} C_VEL
LIN {X 0,Y 171.46,Z 405.119,A -85,B 0,C 180,E1 -23065.612,E2 -23065.612} C_VEL
LIN {X 0,Y 171.439,Z 405.126,A -85,B 0,C 180,E1 -23070.587,E2 -23070.587} C_VEL
LIN {X 0,Y 171.435,Z 405.284,A -85,B 0,C 180,E1 -23075.384,E2 -23075.384} C_VEL
LIN {X 0,Y 172.177,Z 407.394,A -85,B 0,C 180,E1 -23077.202,E2 -23077.202} C_VEL
LIN {X 0,Y 174.263,Z 411.108,A -85,B 0,C 180,E1 -23078.329,E2 -23078.329} C_VEL
LIN {X 0,Y 176.379,Z 413.97,A -85,B 0,C 180,E1 -23079.363,E2 -23079.363} C_VEL
LIN {X 0,Y 180.289,Z 420.239,A -85,B 0,C 180,E1 -23081.213,E2 -23081.213} C_VEL
LIN {X 0,Y 185.2,Z 428.558,A -85,B 0,C 180,E1 -23083.365,E2 -23083.365} C_VEL
LIN {X 0,Y 192.242,Z 442.247,A -85,B 0,C 180,E1 -23086.221,E2 -23086.221} C_VEL
LIN {X 0,Y 198.528,Z 456.956,A -85,B 0,C 180,E1 -23088.617,E2 -23088.617} C_VEL
LIN {X 0,Y 200.547,Z 462.403,A -85,B 0,C 180,E1 -23089.37,E2 -23089.37} C_VEL
LIN {X 0,Y 201.613,Z 472.274,A -85,B 0,C 180,E1 -23090.076,E2 -23090.076} C_VEL
LIN {X 0,Y 199.176,Z 517.377,A -85,B 0,C 180,E1 -23091.62,E2 -23091.62} C_VEL
LIN {X 0,Y 197.428,Z 531.006,A -85,B 0,C 180,E1 -23092.407,E2 -23092.407} C_VEL
LIN {X 0,Y 195.055,Z 543.721,A -85,B 0,C 180,E1 -23093.523,E2 -23093.523} C_VEL
LIN {X 0,Y 192.346,Z 554.803,A -85,B 0,C 180,E1 -23094.868,E2 -23094.868} C_VEL
LIN {X 0,Y 190.103,Z 562.779,A -85,B 0,C 180,E1 -23096.1,E2 -23096.1} C_VEL
LIN {X 0,Y 187.993,Z 567.701,A -85,B 0,C 180,E1 -23096.862,E2 -23096.862} C_VEL
LIN {X 0,Y 182.923,Z 575.353,A -85,B 0,C 180,E1 -23098.028,E2 -23098.028} C_VEL
LIN {X 0,Y 177.723,Z 582.53,A -85,B 0,C 180,E1 -23099.444,E2 -23099.444} C_VEL
LIN {X 0,Y 175.449,Z 586.653,A -85,B 0,C 180,E1 -23100.593,E2 -23100.593} C_VEL
LIN {X 0,Y 171.689,Z 595.689,A -85,B 0,C 180,E1 -23103.916,E2 -23103.916} C_VEL
LIN {X 0,Y 168.705,Z 602.842,A -85,B 0,C 180,E1 -23107.336,E2 -23107.336} C_VEL
LIN {X 0,Y 166.504,Z 607.703,A -85,B 0,C 180,E1 -23110.265,E2 -23110.265} C_VEL
LIN {X 0,Y 164.342,Z 612.427,A -85,B 0,C 180,E1 -23113.861,E2 -23113.861} C_VEL
LIN {X 0,Y 162.984,Z 616.05,A -85,B 0,C 180,E1 -23117.549,E2 -23117.549} C_VEL
LIN {X 0,Y 162.385,Z 617.92,A -85,B 0,C 180,E1 -23120.031,E2 -23120.031} C_VEL
LIN {X 0,Y 161.848,Z 620.332,A -85,B 0,C 180,E1 -23125.018,E2 -23125.018} C_VEL
LIN {X 0,Y 161.839,Z 620.948,A -85,B 0,C 180,E1 -23127.511,E2 -23127.511} C_VEL
LIN {X 0,Y 161.995,Z 621.167,A -85,B 0,C 180,E1 -23130,E2 -23130} C_VEL
LIN {X 0,Y 161.855,Z 620.849,A -85,B 0,C 180,E1 -23132.922,E2 -23132.922} C_VEL
LIN {X 0,Y 161.994,Z 619.293,A -85,B 0,C 180,E1 -23137.478,E2 -23137.478} C_VEL
LIN {X 0,Y 162.382,Z 617.875,A -85,B 0,C 180,E1 -23139.969,E2 -23139.969} C_VEL
LIN {X 0,Y 163.361,Z 614.905,A -85,B 0,C 180,E1 -23143.687,E2 -23143.687} C_VEL
LIN {X 0,Y 164.969,Z 610.9,A -85,B 0,C 180,E1 -23147.35,E2 -23147.35} C_VEL
LIN {X 0,Y 167.7,Z 604.754,A -85,B 0,C 180,E1 -23151.512,E2 -23151.512} C_VEL
LIN {X 0,Y 170.216,Z 599.293,A -85,B 0,C 180,E1 -23154.386,E2 -23154.386} C_VEL
LIN {X 0,Y 173.505,Z 591.23,A -85,B 0,C 180,E1 -23157.763,E2 -23157.763} C_VEL
LIN {X 0,Y 176.891,Z 583.028,A -85,B 0,C 180,E1 -23160.435,E2 -23160.435} C_VEL
LIN {X 0,Y 180.671,Z 573.03,A -85,B 0,C 180,E1 -23162.996,E2 -23162.996} C_VEL
LIN {X 0,Y 184.391,Z 561.729,A -85,B 0,C 180,E1 -23165.203,E2 -23165.203} C_VEL
LIN {X 0,Y 187.5,Z 550.659,A -85,B 0,C 180,E1 -23166.849,E2 -23166.849} C_VEL
LIN {X 0,Y 190.312,Z 538.375,A -85,B 0,C 180,E1 -23168.21,E2 -23168.21} C_VEL
LIN {X 0,Y 192.576,Z 524.83,A -85,B 0,C 180,E1 -23169.234,E2 -23169.234} C_VEL
LIN {X 0,Y 193.885,Z 511.992,A -85,B 0,C 180,E1 -23169.849,E2 -23169.849} C_VEL
LIN {X 0,Y 196.014,Z 473.417,A -85,B 0,C 180,E1 -23171.154,E2 -23171.154} C_VEL
LIN {X 0,Y 194.989,Z 464.113,A -85,B 0,C 180,E1 -23171.862,E2 -23171.862} C_VEL
LIN {X 0,Y 188.557,Z 448.266,A -85,B 0,C 180,E1 -23174.438,E2 -23174.438} C_VEL
LIN {X 0,Y 183.194,Z 437.158,A -85,B 0,C 180,E1 -23176.705,E2 -23176.705} C_VEL
LIN {X 0,Y 177.418,Z 426.819,A -85,B 0,C 180,E1 -23179.324,E2 -23179.324} C_VEL
LIN {X 0,Y 174.717,Z 422.386,A -85,B 0,C 180,E1 -23180.634,E2 -23180.634} C_VEL
LIN {X 0,Y 171.778,Z 417.685,A -85,B 0,C 180,E1 -23182.142,E2 -23182.142} C_VEL
LIN {X 0,Y 168.43,Z 412.535,A -85,B 0,C 180,E1 -23183.979,E2 -23183.979} C_VEL
LIN {X 0,Y 164.999,Z 408.244,A -85,B 0,C 180,E1 -23185.956,E2 -23185.956} C_VEL
LIN {X 0,Y 164.462,Z 406.687,A -85,B 0,C 180,E1 -23186.427,E2 -23186.427} C_VEL
LIN {X 0,Y 164.371,Z 405.998,A -85,B 0,C 180,E1 -23187.273,E2 -23187.273} C_VEL
LIN {X 0,Y 164.34,Z 405.998,A -85,B 0,C 180,E1 -23191.939,E2 -23191.939} C_VEL
LIN {X 0,Y 164.414,Z 405.997,A -85,B 0,C 180,E1 -23194.694,E2 -23194.694} C_VEL
LIN {X 0,Y 164.482,Z 405.995,A -85,B 0,C 180,E1 -23200.051,E2 -23200.051} C_VEL
LIN {X 0,Y 164.521,Z 405.986,A -85,B 0,C 180,E1 -23205.149,E2 -23205.149} C_VEL
LIN {X 0,Y 164.793,Z 405.935,A -85,B 0,C 180,E1 -23210.178,E2 -23210.178} C_VEL
LIN {X 0,Y 164.843,Z 405.95,A -85,B 0,C 180,E1 -23212.652,E2 -23212.652} C_VEL
LIN {X 0,Y 165.046,Z 405.902,A -85,B 0,C 180,E1 -23217.56,E2 -23217.56} C_VEL
LIN {X 0,Y 165.293,Z 405.893,A -85,B 0,C 180,E1 -23220,E2 -23220} C_VEL
LIN {X 0,Y 164.83,Z 405.944,A -85,B 0,C 180,E1 -23227.114,E2 -23227.114} C_VEL
LIN {X 0,Y 164.74,Z 405.944,A -85,B 0,C 180,E1 -23231.132,E2 -23231.132} C_VEL
LIN {X 0,Y 164.48,Z 405.987,A -85,B 0,C 180,E1 -23237.404,E2 -23237.404} C_VEL
LIN {X 0,Y 164.471,Z 405.977,A -85,B 0,C 180,E1 -23239.99,E2 -23239.99} C_VEL
LIN {X 0,Y 164.386,Z 405.99,A -85,B 0,C 180,E1 -23246.131,E2 -23246.131} C_VEL
LIN {X 0,Y 164.374,Z 405.995,A -85,B 0,C 180,E1 -23251.229,E2 -23251.229} C_VEL
LIN {X 0,Y 164.351,Z 406.013,A -85,B 0,C 180,E1 -23254.087,E2 -23254.087} C_VEL
LIN {X 0,Y 165.177,Z 408.515,A -85,B 0,C 180,E1 -23254.73,E2 -23254.73} C_VEL
LIN {X 0,Y 166.983,Z 410.679,A -85,B 0,C 180,E1 -23255.78,E2 -23255.78} C_VEL
LIN {X 0,Y 168.347,Z 411.802,A -85,B 0,C 180,E1 -23256.506,E2 -23256.506} C_VEL
LIN {X 0,Y 170.516,Z 415.198,A -85,B 0,C 180,E1 -23257.72,E2 -23257.72} C_VEL
LIN {X 0,Y 172.129,Z 416.922,A -85,B 0,C 180,E1 -23258.53,E2 -23258.53} C_VEL
LIN {X 0,Y 174.783,Z 420.592,A -85,B 0,C 180,E1 -23259.854,E2 -23259.854} C_VEL
LIN {X 0,Y 180.874,Z 429.522,A -85,B 0,C 180,E1 -23262.653,E2 -23262.653} C_VEL
LIN {X 0,Y 187.391,Z 439.968,A -85,B 0,C 180,E1 -23265.351,E2 -23265.351} C_VEL
LIN {X 0,Y 192.88,Z 449.913,A -85,B 0,C 180,E1 -23267.452,E2 -23267.452} C_VEL
LIN {X 0,Y 196.825,Z 459.079,A -85,B 0,C 180,E1 -23268.946,E2 -23268.946} C_VEL
LIN {X 0,Y 194.058,Z 505.556,A -85,B 0,C 180,E1 -23270.521,E2 -23270.521} C_VEL
LIN {X 0,Y 192.398,Z 519.302,A -85,B 0,C 180,E1 -23271.357,E2 -23271.357} C_VEL
LIN {X 0,Y 190.176,Z 532.363,A -85,B 0,C 180,E1 -23272.596,E2 -23272.596} C_VEL
LIN {X 0,Y 187.443,Z 544.141,A -85,B 0,C 180,E1 -23274.138,E2 -23274.138} C_VEL
LIN {X 0,Y 184.179,Z 555.462,A -85,B 0,C 180,E1 -23276.079,E2 -23276.079} C_VEL
LIN {X 0,Y 180.723,Z 565.661,A -85,B 0,C 180,E1 -23278.333,E2 -23278.333} C_VEL
LIN {X 0,Y 177.238,Z 575.098,A -85,B 0,C 180,E1 -23281.057,E2 -23281.057} C_VEL
LIN {X 0,Y 173.631,Z 583.695,A -85,B 0,C 180,E1 -23284.207,E2 -23284.207} C_VEL
LIN {X 0,Y 170.369,Z 590.849,A -85,B 0,C 180,E1 -23287.569,E2 -23287.569} C_VEL
LIN {X 0,Y 168.065,Z 595.669,A -85,B 0,C 180,E1 -23290.456,E2 -23290.456} C_VEL
LIN {X 0,Y 165.821,Z 600.35,A -85,B 0,C 180,E1 -23294.009,E2 -23294.009} C_VEL
LIN {X 0,Y 164.105,Z 603.929,A -85,B 0,C 180,E1 -23297.636,E2 -23297.636} C_VEL
LIN {X 0,Y 163.305,Z 605.774,A -85,B 0,C 180,E1 -23300.088,E2 -23300.088} C_VEL
LIN {X 0,Y 162.399,Z 607.966,A -85,B 0,C 180,E1 -23304.475,E2 -23304.475} C_VEL
LIN {X 0,Y 162.11,Z 608.747,A -85,B 0,C 180,E1 -23307.515,E2 -23307.515} C_VEL
LIN {X 0,Y 162.06,Z 608.972,A -85,B 0,C 180,E1 -23310,E2 -23310} C_VEL
LIN {X 0,Y 162.11,Z 608.778,A -85,B 0,C 180,E1 -23312.485,E2 -23312.485} C_VEL
LIN {X 0,Y 162.756,Z 607.228,A -85,B 0,C 180,E1 -23317.443,E2 -23317.443} C_VEL
LIN {X 0,Y 163.31,Z 605.876,A -85,B 0,C 180,E1 -23319.912,E2 -23319.912} C_VEL
LIN {X 0,Y 164.623,Z 603.014,A -85,B 0,C 180,E1 -23323.58,E2 -23323.58} C_VEL
LIN {X 0,Y 166.464,Z 599.13,A -85,B 0,C 180,E1 -23327.189,E2 -23327.189} C_VEL
LIN {X 0,Y 168.854,Z 594.117,A -85,B 0,C 180,E1 -23330.718,E2 -23330.718} C_VEL
LIN {X 0,Y 171.829,Z 587.796,A -85,B 0,C 180,E1 -23334.142,E2 -23334.142} C_VEL
LIN {X 0,Y 175.442,Z 579.882,A -85,B 0,C 180,E1 -23337.43,E2 -23337.43} C_VEL
LIN {X 0,Y 178.612,Z 571.613,A -85,B 0,C 180,E1 -23340.188,E2 -23340.188} C_VEL
LIN {X 0,Y 182.09,Z 561.979,A -85,B 0,C 180,E1 -23342.707,E2 -23342.707} C_VEL
LIN {X 0,Y 185.684,Z 550.881,A -85,B 0,C 180,E1 -23344.922,E2 -23344.922} C_VEL
LIN {X 0,Y 188.658,Z 539.999,A -85,B 0,C 180,E1 -23346.586,E2 -23346.586} C_VEL
LIN {X 0,Y 191.2,Z 527.969,A -85,B 0,C 180,E1 -23348.001,E2 -23348.001} C_VEL
LIN {X 0,Y 193.163,Z 515.508,A -85,B 0,C 180,E1 -23349.046,E2 -23349.046} C_VEL
LIN {X 0,Y 194.427,Z 502.792,A -85,B 0,C 180,E1 -23349.733,E2 -23349.733} C_VEL
LIN {X 0,Y 196.991,Z 459.192,A -85,B 0,C 180,E1 -23351.184,E2 -23351.184} C_VEL
LIN {X 0,Y 192.704,Z 449.448,A -85,B 0,C 180,E1 -23352.804,E2 -23352.804} C_VEL
LIN {X 0,Y 186.849,Z 438.94,A -85,B 0,C 180,E1 -23355.064,E2 -23355.064} C_VEL
LIN {X 0,Y 179.93,Z 428.084,A -85,B 0,C 180,E1 -23357.97,E2 -23357.97} C_VEL
LIN {X 0,Y 176.787,Z 423.545,A -85,B 0,C 180,E1 -23359.401,E2 -23359.401} C_VEL
LIN {X 0,Y 174.248,Z 419.987,A -85,B 0,C 180,E1 -23360.621,E2 -23360.621} C_VEL
LIN {X 0,Y 171.435,Z 416.068,A -85,B 0,C 180,E1 -23362.053,E2 -23362.053} C_VEL
LIN {X 0,Y 168.955,Z 413.013,A -85,B 0,C 180,E1 -23363.369,E2 -23363.369} C_VEL
LIN {X 0,Y 167.957,Z 411.329,A -85,B 0,C 180,E1 -23363.954,E2 -23363.954} C_VEL
LIN {X 0,Y 165.714,Z 409.372,A -85,B 0,C 180,E1 -23365.19,E2 -23365.19} C_VEL
LIN {X 0,Y 164.498,Z 406.89,A -85,B 0,C 180,E1 -23366,E2 -23366} C_VEL
LIN {X 0,Y 164.334,Z 406.005,A -85,B 0,C 180,E1 -23366.223,E2 -23366.223} C_VEL
LIN {X 0,Y 164.403,Z 406.007,A -85,B 0,C 180,E1 -23369.137,E2 -23369.137} C_VEL
LIN {X 0,Y 164.414,Z 406.003,A -85,B 0,C 180,E1 -23374.693,E2 -23374.693} C_VEL
LIN {X 0,Y 164.482,Z 405.996,A -85,B 0,C 180,E1 -23380.05,E2 -23380.05} C_VEL
LIN {X 0,Y 164.521,Z 405.99,A -85,B 0,C 180,E1 -23385.149,E2 -23385.149} C_VEL
LIN {X 0,Y 164.799,Z 405.944,A -85,B 0,C 180,E1 -23390.178,E2 -23390.178} C_VEL
LIN {X 0,Y 164.847,Z 405.951,A -85,B 0,C 180,E1 -23392.652,E2 -23392.652} C_VEL
LIN {X 0,Y 165.045,Z 405.92,A -85,B 0,C 180,E1 -23397.559,E2 -23397.559} C_VEL
LIN {X 0,Y 165.293,Z 405.889,A -85,B 0,C 180,E1 -23400,E2 -23400} C_VEL
LIN {X 0,Y 164.769,Z 405.959,A -85,B 0,C 180,E1 -23404.894,E2 -23404.894} C_VEL
LIN {X 0,Y 164.843,Z 405.937,A -85,B 0,C 180,E1 -23407.348,E2 -23407.348} C_VEL
LIN {X 0,Y 164.748,Z 405.962,A -85,B 0,C 180,E1 -23411.146,E2 -23411.146} C_VEL
LIN {X 0,Y 164.483,Z 405.996,A -85,B 0,C 180,E1 -23417.403,E2 -23417.403} C_VEL
LIN {X 0,Y 164.471,Z 405.984,A -85,B 0,C 180,E1 -23419.989,E2 -23419.989} C_VEL
LIN {X 0,Y 164.386,Z 406.003,A -85,B 0,C 180,E1 -23426.131,E2 -23426.131} C_VEL
LIN {X 0,Y 164.38,Z 405.999,A -85,B 0,C 180,E1 -23432.375,E2 -23432.375} C_VEL
LIN {X 0,Y 164.374,Z 406.319,A -85,B 0,C 180,E1 -23433.069,E2 -23433.069} C_VEL
LIN {X 0,Y 164.542,Z 407.083,A -85,B 0,C 180,E1 -23433.554,E2 -23433.554} C_VEL
LIN {X 0,Y 165.814,Z 409.537,A -85,B 0,C 180,E1 -23434.389,E2 -23434.389} C_VEL
LIN {X 0,Y 169.191,Z 413.572,A -85,B 0,C 180,E1 -23436.294,E2 -23436.294} C_VEL
LIN {X 0,Y 172.084,Z 418.03,A -85,B 0,C 180,E1 -23437.871,E2 -23437.871} C_VEL
LIN {X 0,Y 176.762,Z 425.675,A -85,B 0,C 180,E1 -23440.236,E2 -23440.236} C_VEL
LIN {X 0,Y 181.33,Z 433.561,A -85,B 0,C 180,E1 -23442.353,E2 -23442.353} C_VEL
LIN {X 0,Y 187.913,Z 446.691,A -85,B 0,C 180,E1 -23445.187,E2 -23445.187} C_VEL
LIN {X 0,Y 194.071,Z 461.581,A -85,B 0,C 180,E1 -23447.683,E2 -23447.683} C_VEL
LIN {X 0,Y 195.345,Z 465.233,A -85,B 0,C 180,E1 -23448.196,E2 -23448.196} C_VEL
LIN {X 0,Y 196.116,Z 474.497,A -85,B 0,C 180,E1 -23448.836,E2 -23448.836} C_VEL
LIN {X 0,Y 193.621,Z 517.551,A -85,B 0,C 180,E1 -23450.338,E2 -23450.338} C_VEL
LIN {X 0,Y 191.742,Z 531.465,A -85,B 0,C 180,E1 -23451.166,E2 -23451.166} C_VEL
LIN {X 0,Y 189.389,Z 543.46,A -85,B 0,C 180,E1 -23452.245,E2 -23452.245} C_VEL
LIN {X 0,Y 186.13,Z 556.124,A -85,B 0,C 180,E1 -23453.846,E2 -23453.846} C_VEL
LIN {X 0,Y 182.7,Z 567.397,A -85,B 0,C 180,E1 -23455.766,E2 -23455.766} C_VEL
LIN {X 0,Y 179.082,Z 577.553,A -85,B 0,C 180,E1 -23458.009,E2 -23458.009} C_VEL
LIN {X 0,Y 175.449,Z 586.653,A -85,B 0,C 180,E1 -23460.593,E2 -23460.593} C_VEL
LIN {X 0,Y 173.201,Z 590.627,A -85,B 0,C 180,E1 -23461.837,E2 -23461.837} C_VEL
LIN {X 0,Y 168.038,Z 596.636,A -85,B 0,C 180,E1 -23463.848,E2 -23463.848} C_VEL
LIN {X 0,Y 162.966,Z 602.01,A -85,B 0,C 180,E1 -23466.133,E2 -23466.133} C_VEL
LIN {X 0,Y 160.915,Z 604.976,A -85,B 0,C 180,E1 -23467.781,E2 -23467.781} C_VEL
LIN {X 0,Y 158.199,Z 610.723,A -85,B 0,C 180,E1 -23471.882,E2 -23471.882} C_VEL
LIN {X 0,Y 156.437,Z 614.703,A -85,B 0,C 180,E1 -23475.695,E2 -23475.695} C_VEL
LIN {X 0,Y 155.383,Z 617.653,A -85,B 0,C 180,E1 -23479.577,E2 -23479.577} C_VEL
LIN {X 0,Y 154.752,Z 620.064,A -85,B 0,C 180,E1 -23484.789,E2 -23484.789} C_VEL
LIN {X 0,Y 154.747,Z 620.728,A -85,B 0,C 180,E1 -23487.646,E2 -23487.646} C_VEL
LIN {X 0,Y 154.903,Z 620.9,A -85,B 0,C 180,E1 -23490,E2 -23490} C_VEL
LIN {X 0,Y 154.776,Z 620.668,A -85,B 0,C 180,E1 -23492.602,E2 -23492.602} C_VEL
LIN {X 0,Y 154.757,Z 620.041,A -85,B 0,C 180,E1 -23495.211,E2 -23495.211} C_VEL
LIN {X 0,Y 154.943,Z 619.025,A -85,B 0,C 180,E1 -23497.821,E2 -23497.821} C_VEL
LIN {X 0,Y 155.352,Z 617.605,A -85,B 0,C 180,E1 -23500.425,E2 -23500.425} C_VEL
LIN {X 0,Y 156.436,Z 614.636,A -85,B 0,C 180,E1 -23504.305,E2 -23504.305} C_VEL
LIN {X 0,Y 158.192,Z 610.631,A -85,B 0,C 180,E1 -23508.118,E2 -23508.118} C_VEL
LIN {X 0,Y 161.097,Z 604.484,A -85,B 0,C 180,E1 -23512.44,E2 -23512.44} C_VEL
LIN {X 0,Y 164.19,Z 597.844,A -85,B 0,C 180,E1 -23515.988,E2 -23515.988} C_VEL
LIN {X 0,Y 167.891,Z 589.466,A -85,B 0,C 180,E1 -23519.462,E2 -23519.462} C_VEL
LIN {X 0,Y 171.537,Z 580.95,A -85,B 0,C 180,E1 -23522.182,E2 -23522.182} C_VEL
LIN {X 0,Y 175.595,Z 570.434,A -85,B 0,C 180,E1 -23524.773,E2 -23524.773} C_VEL
LIN {X 0,Y 179.092,Z 560.029,A -85,B 0,C 180,E1 -23526.758,E2 -23526.758} C_VEL
LIN {X 0,Y 182.348,Z 548.614,A -85,B 0,C 180,E1 -23528.424,E2 -23528.424} C_VEL
LIN {X 0,Y 185.038,Z 536.851,A -85,B 0,C 180,E1 -23529.684,E2 -23529.684} C_VEL
LIN {X 0,Y 187.263,Z 523.45,A -85,B 0,C 180,E1 -23530.681,E2 -23530.681} C_VEL
LIN {X 0,Y 188.524,Z 511.107,A -85,B 0,C 180,E1 -23531.258,E2 -23531.258} C_VEL
LIN {X 0,Y 190.659,Z 474.567,A -85,B 0,C 180,E1 -23532.504,E2 -23532.504} C_VEL
LIN {X 0,Y 189.843,Z 466.885,A -85,B 0,C 180,E1 -23533.115,E2 -23533.115} C_VEL
LIN {X 0,Y 183.928,Z 451.959,A -85,B 0,C 180,E1 -23535.654,E2 -23535.654} C_VEL
LIN {X 0,Y 178.796,Z 441.233,A -85,B 0,C 180,E1 -23537.968,E2 -23537.968} C_VEL
LIN {X 0,Y 173.808,Z 431.978,A -85,B 0,C 180,E1 -23540.387,E2 -23540.387} C_VEL
LIN {X 0,Y 168.705,Z 423.389,A -85,B 0,C 180,E1 -23543.096,E2 -23543.096} C_VEL
LIN {X 0,Y 165.16,Z 418.001,A -85,B 0,C 180,E1 -23545.145,E2 -23545.145} C_VEL
LIN {X 0,Y 161.929,Z 413.698,A -85,B 0,C 180,E1 -23547.144,E2 -23547.144} C_VEL
LIN {X 0,Y 161.121,Z 412.291,A -85,B 0,C 180,E1 -23547.701,E2 -23547.701} C_VEL
LIN {X 0,Y 158.894,Z 410.485,A -85,B 0,C 180,E1 -23549.134,E2 -23549.134} C_VEL
LIN {X 0,Y 157.563,Z 408.077,A -85,B 0,C 180,E1 -23550.158,E2 -23550.158} C_VEL
LIN {X 0,Y 157.299,Z 406.876,A -85,B 0,C 180,E1 -23550.471,E2 -23550.471} C_VEL
LIN {X 0,Y 157.319,Z 406.883,A -85,B 0,C 180,E1 -23553.466,E2 -23553.466} C_VEL
LIN {X 0,Y 157.392,Z 406.879,A -85,B 0,C 180,E1 -23559.667,E2 -23559.667} C_VEL
LIN {X 0,Y 157.45,Z 406.857,A -85,B 0,C 180,E1 -23564.466,E2 -23564.466} C_VEL
LIN {X 0,Y 157.722,Z 406.815,A -85,B 0,C 180,E1 -23569.733,E2 -23569.733} C_VEL
LIN {X 0,Y 157.8,Z 406.823,A -85,B 0,C 180,E1 -23572.322,E2 -23572.322} C_VEL
LIN {X 0,Y 158.255,Z 406.768,A -85,B 0,C 180,E1 -23580,E2 -23580} C_VEL
LIN {X 0,Y 157.807,Z 406.824,A -85,B 0,C 180,E1 -23587.678,E2 -23587.678} C_VEL
LIN {X 0,Y 157.67,Z 406.823,A -85,B 0,C 180,E1 -23591.302,E2 -23591.302} C_VEL
LIN {X 0,Y 157.451,Z 406.873,A -85,B 0,C 180,E1 -23595.535,E2 -23595.535} C_VEL
LIN {X 0,Y 157.367,Z 406.866,A -85,B 0,C 180,E1 -23600.933,E2 -23600.933} C_VEL
LIN {X 0,Y 157.308,Z 406.872,A -85,B 0,C 180,E1 -23606.682,E2 -23606.682} C_VEL
LIN {X 0,Y 157.328,Z 406.962,A -85,B 0,C 180,E1 -23610.169,E2 -23610.169} C_VEL
LIN {X 0,Y 158.176,Z 409.434,A -85,B 0,C 180,E1 -23610.916,E2 -23610.916} C_VEL
LIN {X 0,Y 159.997,Z 411.633,A -85,B 0,C 180,E1 -23612.184,E2 -23612.184} C_VEL
LIN {X 0,Y 161.521,Z 412.788,A -85,B 0,C 180,E1 -23613.135,E2 -23613.135} C_VEL
LIN {X 0,Y 163.574,Z 416.046,A -85,B 0,C 180,E1 -23614.483,E2 -23614.483} C_VEL
LIN {X 0,Y 165.577,Z 418.136,A -85,B 0,C 180,E1 -23615.644,E2 -23615.644} C_VEL
LIN {X 0,Y 168.158,Z 421.699,A -85,B 0,C 180,E1 -23617.114,E2 -23617.114} C_VEL
LIN {X 0,Y 169.798,Z 423.985,A -85,B 0,C 180,E1 -23618.002,E2 -23618.002} C_VEL
LIN {X 0,Y 172.677,Z 428.024,A -85,B 0,C 180,E1 -23619.482,E2 -23619.482} C_VEL
LIN {X 0,Y 177.523,Z 435.27,A -85,B 0,C 180,E1 -23621.798,E2 -23621.798} C_VEL
LIN {X 0,Y 183.677,Z 445.411,A -85,B 0,C 180,E1 -23624.483,E2 -23624.483} C_VEL
LIN {X 0,Y 188.737,Z 454.906,A -85,B 0,C 180,E1 -23626.533,E2 -23626.533} C_VEL
LIN {X 0,Y 191.363,Z 461.023,A -85,B 0,C 180,E1 -23627.588,E2 -23627.588} C_VEL
LIN {X 0,Y 188.648,Z 505.801,A -85,B 0,C 180,E1 -23629.151,E2 -23629.151} C_VEL
LIN {X 0,Y 186.973,Z 519.271,A -85,B 0,C 180,E1 -23629.98,E2 -23629.98} C_VEL
LIN {X 0,Y 184.826,Z 531.557,A -85,B 0,C 180,E1 -23631.142,E2 -23631.142} C_VEL
LIN {X 0,Y 182.23,Z 542.831,A -85,B 0,C 180,E1 -23632.598,E2 -23632.598} C_VEL
LIN {X 0,Y 178.724,Z 554.448,A -85,B 0,C 180,E1 -23634.549,E2 -23634.549} C_VEL
LIN {X 0,Y 175.091,Z 564.878,A -85,B 0,C 180,E1 -23636.847,E2 -23636.847} C_VEL
LIN {X 0,Y 171.409,Z 574.529,A -85,B 0,C 180,E1 -23639.621,E2 -23639.621} C_VEL
LIN {X 0,Y 167.939,Z 582.617,A -85,B 0,C 180,E1 -23642.592,E2 -23642.592} C_VEL
LIN {X 0,Y 164.342,Z 590.011,A -85,B 0,C 180,E1 -23646.03,E2 -23646.03} C_VEL
LIN {X 0,Y 161.395,Z 595.938,A -85,B 0,C 180,E1 -23649.613,E2 -23649.613} C_VEL
LIN {X 0,Y 158.997,Z 600.619,A -85,B 0,C 180,E1 -23653.303,E2 -23653.303} C_VEL
LIN {X 0,Y 157.184,Z 604.196,A -85,B 0,C 180,E1 -23657.082,E2 -23657.082} C_VEL
LIN {X 0,Y 156.31,Z 606.042,A -85,B 0,C 180,E1 -23659.639,E2 -23659.639} C_VEL
LIN {X 0,Y 155.722,Z 607.424,A -85,B 0,C 180,E1 -23662.219,E2 -23662.219} C_VEL
LIN {X 0,Y 155.028,Z 609.014,A -85,B 0,C 180,E1 -23667.402,E2 -23667.402} C_VEL
LIN {X 0,Y 154.972,Z 609.239,A -85,B 0,C 180,E1 -23670,E2 -23670} C_VEL
LIN {X 0,Y 155.028,Z 609.044,A -85,B 0,C 180,E1 -23672.598,E2 -23672.598} C_VEL
LIN {X 0,Y 155.722,Z 607.495,A -85,B 0,C 180,E1 -23677.781,E2 -23677.781} C_VEL
LIN {X 0,Y 156.314,Z 606.143,A -85,B 0,C 180,E1 -23680.36,E2 -23680.36} C_VEL
LIN {X 0,Y 157.717,Z 603.281,A -85,B 0,C 180,E1 -23684.187,E2 -23684.187} C_VEL
LIN {X 0,Y 159.678,Z 599.397,A -85,B 0,C 180,E1 -23687.944,E2 -23687.944} C_VEL
LIN {X 0,Y 162.236,Z 594.382,A -85,B 0,C 180,E1 -23691.605,E2 -23691.605} C_VEL
LIN {X 0,Y 165.378,Z 588.061,A -85,B 0,C 180,E1 -23695.148,E2 -23695.148} C_VEL
LIN {X 0,Y 169.18,Z 580.146,A -85,B 0,C 180,E1 -23698.536,E2 -23698.536} C_VEL
LIN {X 0,Y 172.601,Z 571.689,A -85,B 0,C 180,E1 -23701.428,E2 -23701.428} C_VEL
LIN {X 0,Y 176.154,Z 562.243,A -85,B 0,C 180,E1 -23703.955,E2 -23703.955} C_VEL
LIN {X 0,Y 179.914,Z 551.144,A -85,B 0,C 180,E1 -23706.215,E2 -23706.215} C_VEL
LIN {X 0,Y 183.017,Z 540.26,A -85,B 0,C 180,E1 -23707.908,E2 -23707.908} C_VEL
LIN {X 0,Y 185.673,Z 528.228,A -85,B 0,C 180,E1 -23709.346,E2 -23709.346} C_VEL
LIN {X 0,Y 187.726,Z 515.662,A -85,B 0,C 180,E1 -23710.415,E2 -23710.415} C_VEL
LIN {X 0,Y 189.054,Z 502.762,A -85,B 0,C 180,E1 -23711.117,E2 -23711.117} C_VEL
LIN {X 0,Y 191.597,Z 461.364,A -85,B 0,C 180,E1 -23712.515,E2 -23712.515} C_VEL
LIN {X 0,Y 187.785,Z 452.761,A -85,B 0,C 180,E1 -23714.049,E2 -23714.049} C_VEL
LIN {X 0,Y 181.204,Z 441.012,A -85,B 0,C 180,E1 -23716.78,E2 -23716.78} C_VEL
LIN {X 0,Y 174.13,Z 430.005,A -85,B 0,C 180,E1 -23720.031,E2 -23720.031} C_VEL
LIN {X 0,Y 170.566,Z 425.062,A -85,B 0,C 180,E1 -23721.825,E2 -23721.825} C_VEL
LIN {X 0,Y 168.11,Z 421.595,A -85,B 0,C 180,E1 -23723.155,E2 -23723.155} C_VEL
LIN {X 0,Y 165.495,Z 417.956,A -85,B 0,C 180,E1 -23724.66,E2 -23724.66} C_VEL
LIN {X 0,Y 162.409,Z 414.48,A -85,B 0,C 180,E1 -23726.514,E2 -23726.514} C_VEL
LIN {X 0,Y 161.196,Z 412.383,A -85,B 0,C 180,E1 -23727.348,E2 -23727.348} C_VEL
LIN {X 0,Y 158.876,Z 410.48,A -85,B 0,C 180,E1 -23728.855,E2 -23728.855} C_VEL
LIN {X 0,Y 157.563,Z 408.029,A -85,B 0,C 180,E1 -23729.881,E2 -23729.881} C_VEL
LIN {X 0,Y 157.302,Z 406.883,A -85,B 0,C 180,E1 -23730.195,E2 -23730.195} C_VEL
LIN {X 0,Y 157.32,Z 406.887,A -85,B 0,C 180,E1 -23733.465,E2 -23733.465} C_VEL
LIN {X 0,Y 157.392,Z 406.881,A -85,B 0,C 180,E1 -23739.667,E2 -23739.667} C_VEL
LIN {X 0,Y 157.451,Z 406.865,A -85,B 0,C 180,E1 -23744.465,E2 -23744.465} C_VEL
LIN {X 0,Y 157.723,Z 406.822,A -85,B 0,C 180,E1 -23749.733,E2 -23749.733} C_VEL
LIN {X 0,Y 157.804,Z 406.829,A -85,B 0,C 180,E1 -23752.322,E2 -23752.322} C_VEL
LIN {X 0,Y 158.255,Z 406.765,A -85,B 0,C 180,E1 -23760,E2 -23760} C_VEL
LIN {X 0,Y 157.781,Z 406.814,A -85,B 0,C 180,E1 -23767.679,E2 -23767.679} C_VEL
LIN {X 0,Y 157.677,Z 406.844,A -85,B 0,C 180,E1 -23771.315,E2 -23771.315} C_VEL
LIN {X 0,Y 157.459,Z 406.859,A -85,B 0,C 180,E1 -23775.534,E2 -23775.534} C_VEL
LIN {X 0,Y 157.367,Z 406.872,A -85,B 0,C 180,E1 -23780.933,E2 -23780.933} C_VEL
LIN {X 0,Y 157.309,Z 406.889,A -85,B 0,C 180,E1 -23786.682,E2 -23786.682} C_VEL
LIN {X 0,Y 157.275,Z 406.904,A -85,B 0,C 180,E1 -23789.35,E2 -23789.35} C_VEL
LIN {X 0,Y 158.105,Z 409.41,A -85,B 0,C 180,E1 -23790.097,E2 -23790.097} C_VEL
LIN {X 0,Y 160.248,Z 411.764,A -85,B 0,C 180,E1 -23791.579,E2 -23791.579} C_VEL
LIN {X 0,Y 161.44,Z 412.58,A -85,B 0,C 180,E1 -23792.32,E2 -23792.32} C_VEL
LIN {X 0,Y 163.278,Z 415.738,A -85,B 0,C 180,E1 -23793.562,E2 -23793.562} C_VEL
LIN {X 0,Y 166.071,Z 419.245,A -85,B 0,C 180,E1 -23795.232,E2 -23795.232} C_VEL
LIN {X 0,Y 170.239,Z 425.885,A -85,B 0,C 180,E1 -23797.605,E2 -23797.605} C_VEL
LIN {X 0,Y 175.285,Z 434.478,A -85,B 0,C 180,E1 -23800.214,E2 -23800.214} C_VEL
LIN {X 0,Y 180.709,Z 444.984,A -85,B 0,C 180,E1 -23802.794,E2 -23802.794} C_VEL
LIN {X 0,Y 185.465,Z 455.476,A -85,B 0,C 180,E1 -23804.909,E2 -23804.909} C_VEL
LIN {X 0,Y 190.122,Z 467.382,A -85,B 0,C 180,E1 -23806.893,E2 -23806.893} C_VEL
LIN {X 0,Y 190.813,Z 474.6,A -85,B 0,C 180,E1 -23807.446,E2 -23807.446} C_VEL
LIN {X 0,Y 188.185,Z 517.12,A -85,B 0,C 180,E1 -23808.938,E2 -23808.938} C_VEL
LIN {X 0,Y 186.33,Z 530.869,A -85,B 0,C 180,E1 -23809.775,E2 -23809.775} C_VEL
LIN {X 0,Y 183.828,Z 543.199,A -85,B 0,C 180,E1 -23810.891,E2 -23810.891} C_VEL
LIN {X 0,Y 180.452,Z 555.862,A -85,B 0,C 180,E1 -23812.517,E2 -23812.517} C_VEL
LIN {X 0,Y 176.873,Z 567.134,A -85,B 0,C 180,E1 -23814.472,E2 -23814.472} C_VEL
LIN {X 0,Y 173.088,Z 577.288,A -85,B 0,C 180,E1 -23816.761,E2 -23816.761} C_VEL
LIN {X 0,Y 169.085,Z 586.852,A -85,B 0,C 180,E1 -23819.565,E2 -23819.565} C_VEL
LIN {X 0,Y 165.321,Z 595.378,A -85,B 0,C 180,E1 -23822.808,E2 -23822.808} C_VEL
LIN {X 0,Y 162.164,Z 602.576,A -85,B 0,C 180,E1 -23826.367,E2 -23826.367} C_VEL
LIN {X 0,Y 160.915,Z 604.976,A -85,B 0,C 180,E1 -23827.781,E2 -23827.781} C_VEL
LIN {X 0,Y 158.938,Z 607.727,A -85,B 0,C 180,E1 -23829.516,E2 -23829.516} C_VEL
LIN {X 0,Y 152.393,Z 612.986,A -85,B 0,C 180,E1 -23833.594,E2 -23833.594} C_VEL
LIN {X 0,Y 149.422,Z 615.392,A -85,B 0,C 180,E1 -23836.228,E2 -23836.228} C_VEL
LIN {X 0,Y 148.691,Z 616.408,A -85,B 0,C 180,E1 -23837.659,E2 -23837.659} C_VEL
LIN {X 0,Y 147.894,Z 618.79,A -85,B 0,C 180,E1 -23841.804,E2 -23841.804} C_VEL
LIN {X 0,Y 147.684,Z 619.797,A -85,B 0,C 180,E1 -23844.539,E2 -23844.539} C_VEL
LIN {X 0,Y 147.663,Z 620.527,A -85,B 0,C 180,E1 -23848.173,E2 -23848.173} C_VEL
LIN {X 0,Y 147.801,Z 620.633,A -85,B 0,C 180,E1 -23850,E2 -23850} C_VEL
LIN {X 0,Y 147.677,Z 620.4,A -85,B 0,C 180,E1 -23852.728,E2 -23852.728} C_VEL
LIN {X 0,Y 147.687,Z 619.774,A -85,B 0,C 180,E1 -23855.461,E2 -23855.461} C_VEL
LIN {X 0,Y 147.89,Z 618.757,A -85,B 0,C 180,E1 -23858.196,E2 -23858.196} C_VEL
LIN {X 0,Y 148.342,Z 617.336,A -85,B 0,C 180,E1 -23860.924,E2 -23860.924} C_VEL
LIN {X 0,Y 149.511,Z 614.366,A -85,B 0,C 180,E1 -23864.983,E2 -23864.983} C_VEL
LIN {X 0,Y 151.421,Z 610.361,A -85,B 0,C 180,E1 -23868.959,E2 -23868.959} C_VEL
LIN {X 0,Y 154.548,Z 604.215,A -85,B 0,C 180,E1 -23873.447,E2 -23873.447} C_VEL
LIN {X 0,Y 157.505,Z 598.192,A -85,B 0,C 180,E1 -23876.821,E2 -23876.821} C_VEL
LIN {X 0,Y 161.006,Z 590.688,A -85,B 0,C 180,E1 -23880.13,E2 -23880.13} C_VEL
LIN {X 0,Y 164.749,Z 582.486,A -85,B 0,C 180,E1 -23882.949,E2 -23882.949} C_VEL
LIN {X 0,Y 168.921,Z 572.488,A -85,B 0,C 180,E1 -23885.624,E2 -23885.624} C_VEL
LIN {X 0,Y 172.991,Z 561.186,A -85,B 0,C 180,E1 -23887.913,E2 -23887.913} C_VEL
LIN {X 0,Y 176.334,Z 550.113,A -85,B 0,C 180,E1 -23889.619,E2 -23889.619} C_VEL
LIN {X 0,Y 179.38,Z 537.827,A -85,B 0,C 180,E1 -23891.014,E2 -23891.014} C_VEL
LIN {X 0,Y 181.763,Z 524.443,A -85,B 0,C 180,E1 -23892.059,E2 -23892.059} C_VEL
LIN {X 0,Y 183.208,Z 511.405,A -85,B 0,C 180,E1 -23892.696,E2 -23892.696} C_VEL
LIN {X 0,Y 185.387,Z 475.057,A -85,B 0,C 180,E1 -23893.974,E2 -23893.974} C_VEL
LIN {X 0,Y 184.773,Z 469.636,A -85,B 0,C 180,E1 -23894.444,E2 -23894.444} C_VEL
LIN {X 0,Y 179.522,Z 456.024,A -85,B 0,C 180,E1 -23896.865,E2 -23896.865} C_VEL
LIN {X 0,Y 174.723,Z 445.675,A -85,B 0,C 180,E1 -23899.184,E2 -23899.184} C_VEL
LIN {X 0,Y 169.949,Z 436.614,A -85,B 0,C 180,E1 -23901.662,E2 -23901.662} C_VEL
LIN {X 0,Y 165.234,Z 428.539,A -85,B 0,C 180,E1 -23904.338,E2 -23904.338} C_VEL
LIN {X 0,Y 161.802,Z 423.189,A -85,B 0,C 180,E1 -23906.465,E2 -23906.465} C_VEL
LIN {X 0,Y 158.921,Z 419.104,A -85,B 0,C 180,E1 -23908.388,E2 -23908.388} C_VEL
LIN {X 0,Y 155.769,Z 415.653,A -85,B 0,C 180,E1 -23910.616,E2 -23910.616} C_VEL
LIN {X 0,Y 154.713,Z 413.51,A -85,B 0,C 180,E1 -23911.512,E2 -23911.512} C_VEL
LIN {X 0,Y 152.296,Z 411.904,A -85,B 0,C 180,E1 -23913.377,E2 -23913.377} C_VEL
LIN {X 0,Y 150.754,Z 409.642,A -85,B 0,C 180,E1 -23914.8,E2 -23914.8} C_VEL
LIN {X 0,Y 150.239,Z 407.753,A -85,B 0,C 180,E1 -23915.471,E2 -23915.471} C_VEL
LIN {X 0,Y 150.357,Z 407.744,A -85,B 0,C 180,E1 -23920.901,E2 -23920.901} C_VEL
LIN {X 0,Y 150.442,Z 407.746,A -85,B 0,C 180,E1 -23926.492,E2 -23926.492} C_VEL
LIN {X 0,Y 150.648,Z 407.696,A -85,B 0,C 180,E1 -23929.245,E2 -23929.245} C_VEL
LIN {X 0,Y 150.735,Z 407.697,A -85,B 0,C 180,E1 -23931.96,E2 -23931.96} C_VEL
LIN {X 0,Y 151.216,Z 407.644,A -85,B 0,C 180,E1 -23940,E2 -23940} C_VEL
LIN {X 0,Y 150.741,Z 407.708,A -85,B 0,C 180,E1 -23948.04,E2 -23948.04} C_VEL
LIN {X 0,Y 150.603,Z 407.701,A -85,B 0,C 180,E1 -23951.492,E2 -23951.492} C_VEL
LIN {X 0,Y 150.36,Z 407.756,A -85,B 0,C 180,E1 -23956.287,E2 -23956.287} C_VEL
LIN {X 0,Y 150.348,Z 407.738,A -85,B 0,C 180,E1 -23960.792,E2 -23960.792} C_VEL
LIN {X 0,Y 150.244,Z 407.806,A -85,B 0,C 180,E1 -23965.16,E2 -23965.16} C_VEL
LIN {X 0,Y 150.929,Z 410.027,A -85,B 0,C 180,E1 -23965.955,E2 -23965.955} C_VEL
LIN {X 0,Y 152.941,Z 412.49,A -85,B 0,C 180,E1 -23967.728,E2 -23967.728} C_VEL
LIN {X 0,Y 154.783,Z 413.658,A -85,B 0,C 180,E1 -23969.124,E2 -23969.124} C_VEL
LIN {X 0,Y 156.714,Z 416.976,A -85,B 0,C 180,E1 -23970.677,E2 -23970.677} C_VEL
LIN {X 0,Y 158.98,Z 419.179,A -85,B 0,C 180,E1 -23972.227,E2 -23972.227} C_VEL
LIN {X 0,Y 161.579,Z 422.817,A -85,B 0,C 180,E1 -23973.963,E2 -23973.963} C_VEL
LIN {X 0,Y 163.063,Z 424.627,A -85,B 0,C 180,E1 -23974.875,E2 -23974.875} C_VEL
LIN {X 0,Y 166.602,Z 429.536,A -85,B 0,C 180,E1 -23976.951,E2 -23976.951} C_VEL
LIN {X 0,Y 171.101,Z 435.998,A -85,B 0,C 180,E1 -23979.353,E2 -23979.353} C_VEL
LIN {X 0,Y 178.063,Z 447.379,A -85,B 0,C 180,E1 -23982.708,E2 -23982.708} C_VEL
LIN {X 0,Y 183.678,Z 457.779,A -85,B 0,C 180,E1 -23985.158,E2 -23985.158} C_VEL
LIN {X 0,Y 186.059,Z 463.176,A -85,B 0,C 180,E1 -23986.175,E2 -23986.175} C_VEL
LIN {X 0,Y 183.382,Z 505.854,A -85,B 0,C 180,E1 -23987.694,E2 -23987.694} C_VEL
LIN {X 0,Y 181.734,Z 518.911,A -85,B 0,C 180,E1 -23988.502,E2 -23988.502} C_VEL
LIN {X 0,Y 179.373,Z 531.831,A -85,B 0,C 180,E1 -23989.724,E2 -23989.724} C_VEL
LIN {X 0,Y 176.662,Z 543.103,A -85,B 0,C 180,E1 -23991.204,E2 -23991.204} C_VEL
LIN {X 0,Y 173.013,Z 554.718,A -85,B 0,C 180,E1 -23993.191,E2 -23993.191} C_VEL
LIN {X 0,Y 169.211,Z 565.148,A -85,B 0,C 180,E1 -23995.536,E2 -23995.536} C_VEL
LIN {X 0,Y 165.596,Z 574.194,A -85,B 0,C 180,E1 -23998.177,E2 -23998.177} C_VEL
LIN {X 0,Y 161.67,Z 582.886,A -85,B 0,C 180,E1 -24001.434,E2 -24001.434} C_VEL
LIN {X 0,Y 157.877,Z 590.28,A -85,B 0,C 180,E1 -24004.983,E2 -24004.983} C_VEL
LIN {X 0,Y 154.745,Z 596.207,A -85,B 0,C 180,E1 -24008.695,E2 -24008.695} C_VEL
LIN {X 0,Y 152.2,Z 600.887,A -85,B 0,C 180,E1 -24012.534,E2 -24012.534} C_VEL
LIN {X 0,Y 150.287,Z 604.464,A -85,B 0,C 180,E1 -24016.478,E2 -24016.478} C_VEL
LIN {X 0,Y 149.343,Z 606.309,A -85,B 0,C 180,E1 -24019.15,E2 -24019.15} C_VEL
LIN {X 0,Y 148.687,Z 607.692,A -85,B 0,C 180,E1 -24021.848,E2 -24021.848} C_VEL
LIN {X 0,Y 147.938,Z 609.281,A -85,B 0,C 180,E1 -24027.277,E2 -24027.277} C_VEL
LIN {X 0,Y 147.885,Z 609.506,A -85,B 0,C 180,E1 -24030,E2 -24030} C_VEL
LIN {X 0,Y 148.124,Z 608.894,A -85,B 0,C 180,E1 -24034.87,E2 -24034.87} C_VEL
LIN {X 0,Y 148.688,Z 607.761,A -85,B 0,C 180,E1 -24038.152,E2 -24038.152} C_VEL
LIN {X 0,Y 149.347,Z 606.409,A -85,B 0,C 180,E1 -24040.849,E2 -24040.849} C_VEL
LIN {X 0,Y 150.841,Z 603.547,A -85,B 0,C 180,E1 -24044.848,E2 -24044.848} C_VEL
LIN {X 0,Y 152.925,Z 599.663,A -85,B 0,C 180,E1 -24048.765,E2 -24048.765} C_VEL
LIN {X 0,Y 155.639,Z 594.648,A -85,B 0,C 180,E1 -24052.57,E2 -24052.57} C_VEL
LIN {X 0,Y 158.985,Z 588.326,A -85,B 0,C 180,E1 -24056.234,E2 -24056.234} C_VEL
LIN {X 0,Y 162.977,Z 580.411,A -85,B 0,C 180,E1 -24059.729,E2 -24059.729} C_VEL
LIN {X 0,Y 166.71,Z 571.637,A -85,B 0,C 180,E1 -24062.802,E2 -24062.802} C_VEL
LIN {X 0,Y 170.737,Z 561.404,A -85,B 0,C 180,E1 -24065.55,E2 -24065.55} C_VEL
LIN {X 0,Y 174.703,Z 549.984,A -85,B 0,C 180,E1 -24067.84,E2 -24067.84} C_VEL
LIN {X 0,Y 177.931,Z 538.761,A -85,B 0,C 180,E1 -24069.561,E2 -24069.561} C_VEL
LIN {X 0,Y 180.493,Z 527.346,A -85,B 0,C 180,E1 -24070.891,E2 -24070.891} C_VEL
LIN {X 0,Y 182.471,Z 515.42,A -85,B 0,C 180,E1 -24071.886,E2 -24071.886} C_VEL
LIN {X 0,Y 183.791,Z 502.849,A -85,B 0,C 180,E1 -24072.575,E2 -24072.575} C_VEL
LIN {X 0,Y 186.265,Z 463.497,A -85,B 0,C 180,E1 -24073.938,E2 -24073.938} C_VEL
LIN {X 0,Y 182.876,Z 455.957,A -85,B 0,C 180,E1 -24075.393,E2 -24075.393} C_VEL
LIN {X 0,Y 176.569,Z 444.732,A -85,B 0,C 180,E1 -24078.196,E2 -24078.196} C_VEL
LIN {X 0,Y 170.791,Z 435.5,A -85,B 0,C 180,E1 -24081.036,E2 -24081.036} C_VEL
LIN {X 0,Y 165.423,Z 427.74,A -85,B 0,C 180,E1 -24083.978,E2 -24083.978} C_VEL
LIN {X 0,Y 162.004,Z 423.195,A -85,B 0,C 180,E1 -24086.045,E2 -24086.045} C_VEL
LIN {X 0,Y 159.378,Z 419.88,A -85,B 0,C 180,E1 -24087.762,E2 -24087.762} C_VEL
LIN {X 0,Y 158.482,Z 418.565,A -85,B 0,C 180,E1 -24088.396,E2 -24088.396} C_VEL
LIN {X 0,Y 156.011,Z 415.976,A -85,B 0,C 180,E1 -24090.154,E2 -24090.154} C_VEL
LIN {X 0,Y 154.625,Z 413.48,A -85,B 0,C 180,E1 -24091.309,E2 -24091.309} C_VEL
LIN {X 0,Y 152.063,Z 411.666,A -85,B 0,C 180,E1 -24093.333,E2 -24093.333} C_VEL
LIN {X 0,Y 150.573,Z 409.22,A -85,B 0,C 180,E1 -24094.767,E2 -24094.767} C_VEL
LIN {X 0,Y 150.249,Z 407.76,A -85,B 0,C 180,E1 -24095.288,E2 -24095.288} C_VEL
LIN {X 0,Y 150.357,Z 407.746,A -85,B 0,C 180,E1 -24100.901,E2 -24100.901} C_VEL
LIN {X 0,Y 150.442,Z 407.742,A -85,B 0,C 180,E1 -24106.492,E2 -24106.492} C_VEL
LIN {X 0,Y 150.645,Z 407.701,A -85,B 0,C 180,E1 -24109.245,E2 -24109.245} C_VEL
LIN {X 0,Y 150.739,Z 407.709,A -85,B 0,C 180,E1 -24111.959,E2 -24111.959} C_VEL
LIN {X 0,Y 151.216,Z 407.641,A -85,B 0,C 180,E1 -24120,E2 -24120} C_VEL
LIN {X 0,Y 150.721,Z 407.691,A -85,B 0,C 180,E1 -24128.041,E2 -24128.041} C_VEL
LIN {X 0,Y 150.608,Z 407.724,A -85,B 0,C 180,E1 -24131.5,E2 -24131.5} C_VEL
LIN {X 0,Y 150.365,Z 407.749,A -85,B 0,C 180,E1 -24136.286,E2 -24136.286} C_VEL
LIN {X 0,Y 150.348,Z 407.745,A -85,B 0,C 180,E1 -24140.792,E2 -24140.792} C_VEL
LIN {X 0,Y 150.261,Z 407.872,A -85,B 0,C 180,E1 -24144.342,E2 -24144.342} C_VEL
LIN {X 0,Y 150.963,Z 410.151,A -85,B 0,C 180,E1 -24145.166,E2 -24145.166} C_VEL
LIN {X 0,Y 152.957,Z 412.502,A -85,B 0,C 180,E1 -24146.933,E2 -24146.933} C_VEL
LIN {X 0,Y 154.821,Z 413.829,A -85,B 0,C 180,E1 -24148.374,E2 -24148.374} C_VEL
LIN {X 0,Y 156.653,Z 416.869,A -85,B 0,C 180,E1 -24149.852,E2 -24149.852} C_VEL
LIN {X 0,Y 158.931,Z 419.082,A -85,B 0,C 180,E1 -24151.427,E2 -24151.427} C_VEL
LIN {X 0,Y 161.362,Z 422.58,A -85,B 0,C 180,E1 -24153.079,E2 -24153.079} C_VEL
LIN {X 0,Y 163.183,Z 425.167,A -85,B 0,C 180,E1 -24154.237,E2 -24154.237} C_VEL
LIN {X 0,Y 166.915,Z 431.294,A -85,B 0,C 180,E1 -24156.494,E2 -24156.494} C_VEL
LIN {X 0,Y 171.436,Z 439.1,A -85,B 0,C 180,E1 -24158.982,E2 -24158.982} C_VEL
LIN {X 0,Y 177.373,Z 451.074,A -85,B 0,C 180,E1 -24161.987,E2 -24161.987} C_VEL
LIN {X 0,Y 181.588,Z 460.988,A -85,B 0,C 180,E1 -24163.986,E2 -24163.986} C_VEL
LIN {X 0,Y 185.17,Z 470.766,A -85,B 0,C 180,E1 -24165.633,E2 -24165.633} C_VEL
LIN {X 0,Y 185.566,Z 475.883,A -85,B 0,C 180,E1 -24166.021,E2 -24166.021} C_VEL
LIN {X 0,Y 182.884,Z 516.935,A -85,B 0,C 180,E1 -24167.48,E2 -24167.48} C_VEL
LIN {X 0,Y 180.95,Z 530.806,A -85,B 0,C 180,E1 -24168.342,E2 -24168.342} C_VEL
LIN {X 0,Y 178.361,Z 542.938,A -85,B 0,C 180,E1 -24169.448,E2 -24169.448} C_VEL
LIN {X 0,Y 174.882,Z 555.601,A -85,B 0,C 180,E1 -24171.104,E2 -24171.104} C_VEL
LIN {X 0,Y 171.128,Z 566.87,A -85,B 0,C 180,E1 -24173.086,E2 -24173.086} C_VEL
LIN {X 0,Y 167.171,Z 577.023,A -85,B 0,C 180,E1 -24175.421,E2 -24175.421} C_VEL
LIN {X 0,Y 163.174,Z 586.177,A -85,B 0,C 180,E1 -24178.156,E2 -24178.156} C_VEL
LIN {X 0,Y 158.937,Z 595.246,A -85,B 0,C 180,E1 -24181.69,E2 -24181.69} C_VEL
LIN {X 0,Y 155.659,Z 602.31,A -85,B 0,C 180,E1 -24185.315,E2 -24185.315} C_VEL
LIN {X 0,Y 153.108,Z 607.167,A -85,B 0,C 180,E1 -24188.456,E2 -24188.456} C_VEL
LIN {X 0,Y 150.679,Z 611.892,A -85,B 0,C 180,E1 -24192.352,E2 -24192.352} C_VEL
LIN {X 0,Y 149.067,Z 615.514,A -85,B 0,C 180,E1 -24196.366,E2 -24196.366} C_VEL
LIN {X 0,Y 148.691,Z 616.408,A -85,B 0,C 180,E1 -24197.659,E2 -24197.659} C_VEL
LIN {X 0,Y 147.525,Z 617.816,A -85,B 0,C 180,E1 -24199.837,E2 -24199.837} C_VEL
LIN {X 0,Y 144.149,Z 619.382,A -85,B 0,C 180,E1 -24203.451,E2 -24203.451} C_VEL
LIN {X 0,Y 141.612,Z 620.069,A -85,B 0,C 180,E1 -24206.479,E2 -24206.479} C_VEL
LIN {X 0,Y 140.685,Z 620.315,A -85,B 0,C 180,E1 -24208.865,E2 -24208.865} C_VEL
LIN {X 0,Y 140.68,Z 620.349,A -85,B 0,C 180,E1 -24209.673,E2 -24209.673} C_VEL
LIN {X 0,Y 140.588,Z 620.133,A -85,B 0,C 180,E1 -24212.865,E2 -24212.865} C_VEL
LIN {X 0,Y 140.615,Z 619.506,A -85,B 0,C 180,E1 -24215.737,E2 -24215.737} C_VEL
LIN {X 0,Y 140.838,Z 618.488,A -85,B 0,C 180,E1 -24218.61,E2 -24218.61} C_VEL
LIN {X 0,Y 141.355,Z 617.067,A -85,B 0,C 180,E1 -24221.471,E2 -24221.471} C_VEL
LIN {X 0,Y 142.621,Z 614.096,A -85,B 0,C 180,E1 -24225.725,E2 -24225.725} C_VEL
LIN {X 0,Y 144.694,Z 610.092,A -85,B 0,C 180,E1 -24229.876,E2 -24229.876} C_VEL
LIN {X 0,Y 148.056,Z 603.946,A -85,B 0,C 180,E1 -24234.541,E2 -24234.541} C_VEL
LIN {X 0,Y 151.517,Z 597.238,A -85,B 0,C 180,E1 -24238.387,E2 -24238.387} C_VEL
LIN {X 0,Y 155.644,Z 588.926,A -85,B 0,C 180,E1 -24242.043,E2 -24242.043} C_VEL
LIN {X 0,Y 159.661,Z 580.408,A -85,B 0,C 180,E1 -24244.905,E2 -24244.905} C_VEL
LIN {X 0,Y 164.116,Z 569.891,A -85,B 0,C 180,E1 -24247.605,E2 -24247.605} C_VEL
LIN {X 0,Y 168.377,Z 558.051,A -85,B 0,C 180,E1 -24249.921,E2 -24249.921} C_VEL
LIN {X 0,Y 171.948,Z 546.118,A -85,B 0,C 180,E1 -24251.618,E2 -24251.618} C_VEL
LIN {X 0,Y 174.904,Z 533.698,A -85,B 0,C 180,E1 -24252.888,E2 -24252.888} C_VEL
LIN {X 0,Y 177.132,Z 520.547,A -85,B 0,C 180,E1 -24253.806,E2 -24253.806} C_VEL
LIN {X 0,Y 178.414,Z 505.534,A -85,B 0,C 180,E1 -24254.453,E2 -24254.453} C_VEL
LIN {X 0,Y 180.271,Z 475.902,A -85,B 0,C 180,E1 -24255.501,E2 -24255.501} C_VEL
LIN {X 0,Y 179.743,Z 472.092,A -85,B 0,C 180,E1 -24255.884,E2 -24255.884} C_VEL
LIN {X 0,Y 174.792,Z 459.123,A -85,B 0,C 180,E1 -24258.342,E2 -24258.342} C_VEL
LIN {X 0,Y 170.383,Z 449.456,A -85,B 0,C 180,E1 -24260.641,E2 -24260.641} C_VEL
LIN {X 0,Y 166.32,Z 441.501,A -85,B 0,C 180,E1 -24262.912,E2 -24262.912} C_VEL
LIN {X 0,Y 161.741,Z 433.477,A -85,B 0,C 180,E1 -24265.7,E2 -24265.7} C_VEL
LIN {X 0,Y 158.821,Z 428.757,A -85,B 0,C 180,E1 -24267.645,E2 -24267.645} C_VEL
LIN {X 0,Y 155.883,Z 424.651,A -85,B 0,C 180,E1 -24269.734,E2 -24269.734} C_VEL
LIN {X 0,Y 153.129,Z 421.351,A -85,B 0,C 180,E1 -24271.844,E2 -24271.844} C_VEL
LIN {X 0,Y 152.125,Z 419.844,A -85,B 0,C 180,E1 -24272.7,E2 -24272.7} C_VEL
LIN {X 0,Y 149.611,Z 417.511,A -85,B 0,C 180,E1 -24274.858,E2 -24274.858} C_VEL
LIN {X 0,Y 147.995,Z 414.466,A -85,B 0,C 180,E1 -24276.565,E2 -24276.565} C_VEL
LIN {X 0,Y 145.456,Z 412.882,A -85,B 0,C 180,E1 -24279.167,E2 -24279.167} C_VEL
LIN {X 0,Y 143.804,Z 410.524,A -85,B 0,C 180,E1 -24281.293,E2 -24281.293} C_VEL
LIN {X 0,Y 143.274,Z 408.615,A -85,B 0,C 180,E1 -24282.331,E2 -24282.331} C_VEL
LIN {X 0,Y 143.592,Z 408.576,A -85,B 0,C 180,E1 -24288.71,E2 -24288.71} C_VEL
LIN {X 0,Y 143.656,Z 408.574,A -85,B 0,C 180,E1 -24291.56,E2 -24291.56} C_VEL
LIN {X 0,Y 144.174,Z 408.52,A -85,B 0,C 180,E1 -24300,E2 -24300} C_VEL
LIN {X 0,Y 143.66,Z 408.591,A -85,B 0,C 180,E1 -24308.44,E2 -24308.44} C_VEL
LIN {X 0,Y 143.546,Z 408.578,A -85,B 0,C 180,E1 -24311.713,E2 -24311.713} C_VEL
LIN {X 0,Y 143.291,Z 408.799,A -85,B 0,C 180,E1 -24318.406,E2 -24318.406} C_VEL
LIN {X 0,Y 144.143,Z 411.223,A -85,B 0,C 180,E1 -24319.771,E2 -24319.771} C_VEL
LIN {X 0,Y 146.259,Z 413.639,A -85,B 0,C 180,E1 -24322.305,E2 -24322.305} C_VEL
LIN {X 0,Y 148.122,Z 414.77,A -85,B 0,C 180,E1 -24324.157,E2 -24324.157} C_VEL
LIN {X 0,Y 149.922,Z 417.931,A -85,B 0,C 180,E1 -24326.01,E2 -24326.01} C_VEL
LIN {X 0,Y 152.69,Z 420.463,A -85,B 0,C 180,E1 -24328.338,E2 -24328.338} C_VEL
LIN {X 0,Y 154.913,Z 423.79,A -85,B 0,C 180,E1 -24330.149,E2 -24330.149} C_VEL
LIN {X 0,Y 156.618,Z 425.635,A -85,B 0,C 180,E1 -24331.379,E2 -24331.379} C_VEL
LIN {X 0,Y 159.459,Z 429.382,A -85,B 0,C 180,E1 -24333.336,E2 -24333.336} C_VEL
LIN {X 0,Y 164.137,Z 436.085,A -85,B 0,C 180,E1 -24336.26,E2 -24336.26} C_VEL
LIN {X 0,Y 168.224,Z 442.258,A -85,B 0,C 180,E1 -24338.555,E2 -24338.555} C_VEL
LIN {X 0,Y 174.323,Z 452.467,A -85,B 0,C 180,E1 -24341.656,E2 -24341.656} C_VEL
LIN {X 0,Y 179.666,Z 462.726,A -85,B 0,C 180,E1 -24344.139,E2 -24344.139} C_VEL
LIN {X 0,Y 180.923,Z 465.614,A -85,B 0,C 180,E1 -24344.712,E2 -24344.712} C_VEL
LIN {X 0,Y 178.134,Z 506.732,A -85,B 0,C 180,E1 -24346.189,E2 -24346.189} C_VEL
LIN {X 0,Y 176.291,Z 520.191,A -85,B 0,C 180,E1 -24347.045,E2 -24347.045} C_VEL
LIN {X 0,Y 173.783,Z 533.182,A -85,B 0,C 180,E1 -24348.338,E2 -24348.338} C_VEL
LIN {X 0,Y 170.696,Z 544.955,A -85,B 0,C 180,E1 -24349.961,E2 -24349.961} C_VEL
LIN {X 0,Y 166.954,Z 556.275,A -85,B 0,C 180,E1 -24352.002,E2 -24352.002} C_VEL
LIN {X 0,Y 162.983,Z 566.472,A -85,B 0,C 180,E1 -24354.4,E2 -24354.4} C_VEL
LIN {X 0,Y 158.855,Z 576.066,A -85,B 0,C 180,E1 -24357.393,E2 -24357.393} C_VEL
LIN {X 0,Y 154.774,Z 584.502,A -85,B 0,C 180,E1 -24360.782,E2 -24360.782} C_VEL
LIN {X 0,Y 150.915,Z 591.656,A -85,B 0,C 180,E1 -24364.485,E2 -24364.485} C_VEL
LIN {X 0,Y 148.141,Z 596.476,A -85,B 0,C 180,E1 -24367.696,E2 -24367.696} C_VEL
LIN {X 0,Y 145.436,Z 601.156,A -85,B 0,C 180,E1 -24371.694,E2 -24371.694} C_VEL
LIN {X 0,Y 143.387,Z 604.732,A -85,B 0,C 180,E1 -24375.814,E2 -24375.814} C_VEL
LIN {X 0,Y 142.367,Z 606.577,A -85,B 0,C 180,E1 -24378.612,E2 -24378.612} C_VEL
LIN {X 0,Y 141.668,Z 607.959,A -85,B 0,C 180,E1 -24381.441,E2 -24381.441} C_VEL
LIN {X 0,Y 140.865,Z 609.548,A -85,B 0,C 180,E1 -24387.14,E2 -24387.14} C_VEL
LIN {X 0,Y 140.818,Z 609.772,A -85,B 0,C 180,E1 -24390,E2 -24390} C_VEL
LIN {X 0,Y 141.01,Z 609.293,A -85,B 0,C 180,E1 -24394.575,E2 -24394.575} C_VEL
LIN {X 0,Y 141.668,Z 608.028,A -85,B 0,C 180,E1 -24398.559,E2 -24398.559} C_VEL
LIN {X 0,Y 142.37,Z 606.676,A -85,B 0,C 180,E1 -24401.388,E2 -24401.388} C_VEL
LIN {X 0,Y 143.998,Z 603.813,A -85,B 0,C 180,E1 -24405.571,E2 -24405.571} C_VEL
LIN {X 0,Y 146.215,Z 599.929,A -85,B 0,C 180,E1 -24409.661,E2 -24409.661} C_VEL
LIN {X 0,Y 149.099,Z 594.914,A -85,B 0,C 180,E1 -24413.619,E2 -24413.619} C_VEL
LIN {X 0,Y 152.652,Z 588.591,A -85,B 0,C 180,E1 -24417.412,E2 -24417.412} C_VEL
LIN {X 0,Y 156.847,Z 580.676,A -85,B 0,C 180,E1 -24421.016,E2 -24421.016} C_VEL
LIN {X 0,Y 160.731,Z 572.033,A -85,B 0,C 180,E1 -24424.13,E2 -24424.13} C_VEL
LIN {X 0,Y 164.579,Z 562.77,A -85,B 0,C 180,E1 -24426.714,E2 -24426.714} C_VEL
LIN {X 0,Y 168.702,Z 551.667,A -85,B 0,C 180,E1 -24429.056,E2 -24429.056} C_VEL
LIN {X 0,Y 172.068,Z 540.781,A -85,B 0,C 180,E1 -24430.806,E2 -24430.806} C_VEL
LIN {X 0,Y 174.961,Z 528.745,A -85,B 0,C 180,E1 -24432.285,E2 -24432.285} C_VEL
LIN {X 0,Y 177.16,Z 516.348,A -85,B 0,C 180,E1 -24433.373,E2 -24433.373} C_VEL
LIN {X 0,Y 178.64,Z 503.081,A -85,B 0,C 180,E1 -24434.113,E2 -24434.113} C_VEL
LIN {X 0,Y 181.076,Z 466.521,A -85,B 0,C 180,E1 -24435.388,E2 -24435.388} C_VEL
LIN {X 0,Y 180.751,Z 464.922,A -85,B 0,C 180,E1 -24435.582,E2 -24435.582} C_VEL
LIN {X 0,Y 176.413,Z 456.131,A -85,B 0,C 180,E1 -24437.572,E2 -24437.572} C_VEL
LIN {X 0,Y 170.26,Z 445.427,A -85,B 0,C 180,E1 -24440.605,E2 -24440.605} C_VEL
LIN {X 0,Y 164.879,Z 437.054,A -85,B 0,C 180,E1 -24443.562,E2 -24443.562} C_VEL
LIN {X 0,Y 159.499,Z 429.408,A -85,B 0,C 180,E1 -24446.909,E2 -24446.909} C_VEL
LIN {X 0,Y 156.659,Z 425.652,A -85,B 0,C 180,E1 -24448.882,E2 -24448.882} C_VEL
LIN {X 0,Y 155.157,Z 424,A -85,B 0,C 180,E1 -24449.973,E2 -24449.973} C_VEL
LIN {X 0,Y 152.723,Z 420.544,A -85,B 0,C 180,E1 -24451.949,E2 -24451.949} C_VEL
LIN {X 0,Y 152.09,Z 419.827,A -85,B 0,C 180,E1 -24452.477,E2 -24452.477} C_VEL
LIN {X 0,Y 149.531,Z 417.416,A -85,B 0,C 180,E1 -24454.711,E2 -24454.711} C_VEL
LIN {X 0,Y 147.982,Z 414.473,A -85,B 0,C 180,E1 -24456.377,E2 -24456.377} C_VEL
LIN {X 0,Y 145.338,Z 412.793,A -85,B 0,C 180,E1 -24459.149,E2 -24459.149} C_VEL
LIN {X 0,Y 143.742,Z 410.358,A -85,B 0,C 180,E1 -24461.285,E2 -24461.285} C_VEL
LIN {X 0,Y 143.268,Z 408.621,A -85,B 0,C 180,E1 -24462.146,E2 -24462.146} C_VEL
LIN {X 0,Y 143.592,Z 408.579,A -85,B 0,C 180,E1 -24468.71,E2 -24468.71} C_VEL
LIN {X 0,Y 143.658,Z 408.588,A -85,B 0,C 180,E1 -24471.56,E2 -24471.56} C_VEL
LIN {X 0,Y 144.174,Z 408.517,A -85,B 0,C 180,E1 -24480,E2 -24480} C_VEL
LIN {X 0,Y 143.645,Z 408.572,A -85,B 0,C 180,E1 -24488.44,E2 -24488.44} C_VEL
LIN {X 0,Y 143.546,Z 408.603,A -85,B 0,C 180,E1 -24491.713,E2 -24491.713} C_VEL
LIN {X 0,Y 143.324,Z 408.826,A -85,B 0,C 180,E1 -24497.478,E2 -24497.478} C_VEL
LIN {X 0,Y 143.976,Z 410.907,A -85,B 0,C 180,E1 -24498.591,E2 -24498.591} C_VEL
LIN {X 0,Y 146.067,Z 413.445,A -85,B 0,C 180,E1 -24501.201,E2 -24501.201} C_VEL
LIN {X 0,Y 148.141,Z 414.785,A -85,B 0,C 180,E1 -24503.318,E2 -24503.318} C_VEL
LIN {X 0,Y 149.72,Z 417.695,A -85,B 0,C 180,E1 -24504.99,E2 -24504.99} C_VEL
LIN {X 0,Y 152.566,Z 420.29,A -85,B 0,C 180,E1 -24507.429,E2 -24507.429} C_VEL
LIN {X 0,Y 154.929,Z 423.755,A -85,B 0,C 180,E1 -24509.372,E2 -24509.372} C_VEL
LIN {X 0,Y 156.488,Z 425.405,A -85,B 0,C 180,E1 -24510.507,E2 -24510.507} C_VEL
LIN {X 0,Y 160.163,Z 430.719,A -85,B 0,C 180,E1 -24513.077,E2 -24513.077} C_VEL
LIN {X 0,Y 163.938,Z 437.123,A -85,B 0,C 180,E1 -24515.507,E2 -24515.507} C_VEL
LIN {X 0,Y 168.137,Z 444.764,A -85,B 0,C 180,E1 -24517.969,E2 -24517.969} C_VEL
LIN {X 0,Y 173.499,Z 456.015,A -85,B 0,C 180,E1 -24520.864,E2 -24520.864} C_VEL
LIN {X 0,Y 177.25,Z 465.097,A -85,B 0,C 180,E1 -24522.766,E2 -24522.766} C_VEL
LIN {X 0,Y 180.22,Z 473.369,A -85,B 0,C 180,E1 -24524.232,E2 -24524.232} C_VEL
LIN {X 0,Y 180.439,Z 477.192,A -85,B 0,C 180,E1 -24524.515,E2 -24524.515} C_VEL
LIN {X 0,Y 177.735,Z 516.683,A -85,B 0,C 180,E1 -24525.939,E2 -24525.939} C_VEL
LIN {X 0,Y 175.764,Z 530.313,A -85,B 0,C 180,E1 -24526.789,E2 -24526.789} C_VEL
LIN {X 0,Y 173.034,Z 542.677,A -85,B 0,C 180,E1 -24527.921,E2 -24527.921} C_VEL
LIN {X 0,Y 169.423,Z 555.339,A -85,B 0,C 180,E1 -24529.598,E2 -24529.598} C_VEL
LIN {X 0,Y 165.49,Z 566.606,A -85,B 0,C 180,E1 -24531.605,E2 -24531.605} C_VEL
LIN {X 0,Y 161.366,Z 576.758,A -85,B 0,C 180,E1 -24533.988,E2 -24533.988} C_VEL
LIN {X 0,Y 157.178,Z 585.912,A -85,B 0,C 180,E1 -24536.789,E2 -24536.789} C_VEL
LIN {X 0,Y 152.761,Z 594.843,A -85,B 0,C 180,E1 -24540.359,E2 -24540.359} C_VEL
LIN {X 0,Y 149.63,Z 601.111,A -85,B 0,C 180,E1 -24543.626,E2 -24543.626} C_VEL
LIN {X 0,Y 146.476,Z 606.899,A -85,B 0,C 180,E1 -24547.428,E2 -24547.428} C_VEL
LIN {X 0,Y 143.901,Z 611.625,A -85,B 0,C 180,E1 -24551.491,E2 -24551.491} C_VEL
LIN {X 0,Y 142.146,Z 615.246,A -85,B 0,C 180,E1 -24555.688,E2 -24555.688} C_VEL
LIN {X 0,Y 141.374,Z 617.117,A -85,B 0,C 180,E1 -24558.531,E2 -24558.531} C_VEL
LIN {X 0,Y 140.614,Z 619.53,A -85,B 0,C 180,E1 -24564.263,E2 -24564.263} C_VEL
LIN {X 0,Y 140.68,Z 620.349,A -85,B 0,C 180,E1 -24569.673,E2 -24569.673} C_VEL
LIN {X 0,Y 140.487,Z 620.357,A -85,B 0,C 180,E1 -24571.268,E2 -24571.268} C_VEL
LIN {X 0,Y 139.729,Z 620.221,A -85,B 0,C 180,E1 -24572.845,E2 -24572.845} C_VEL
LIN {X 0,Y 137.351,Z 619.546,A -85,B 0,C 180,E1 -24575.973,E2 -24575.973} C_VEL
LIN {X 0,Y 135.058,Z 618.321,A -85,B 0,C 180,E1 -24579.191,E2 -24579.191} C_VEL
LIN {X 0,Y 134.361,Z 617.036,A -85,B 0,C 180,E1 -24581.668,E2 -24581.668} C_VEL
LIN {X 0,Y 134.461,Z 616.536,A -85,B 0,C 180,E1 -24582.493,E2 -24582.493} C_VEL
LIN {X 0,Y 136.374,Z 612.586,A -85,B 0,C 180,E1 -24588.011,E2 -24588.011} C_VEL
LIN {X 0,Y 138.952,Z 608.218,A -85,B 0,C 180,E1 -24592.292,E2 -24592.292} C_VEL
LIN {X 0,Y 142.219,Z 602.663,A -85,B 0,C 180,E1 -24596.407,E2 -24596.407} C_VEL
LIN {X 0,Y 145.969,Z 595.728,A -85,B 0,C 180,E1 -24600.367,E2 -24600.367} C_VEL
LIN {X 0,Y 149.646,Z 588.655,A -85,B 0,C 180,E1 -24603.492,E2 -24603.492} C_VEL
LIN {X 0,Y 153.874,Z 580.137,A -85,B 0,C 180,E1 -24606.423,E2 -24606.423} C_VEL
LIN {X 0,Y 158.547,Z 569.62,A -85,B 0,C 180,E1 -24609.172,E2 -24609.172} C_VEL
LIN {X 0,Y 162.503,Z 559.213,A -85,B 0,C 180,E1 -24611.264,E2 -24611.264} C_VEL
LIN {X 0,Y 166.189,Z 547.796,A -85,B 0,C 180,E1 -24612.992,E2 -24612.992} C_VEL
LIN {X 0,Y 169.212,Z 536.026,A -85,B 0,C 180,E1 -24614.288,E2 -24614.288} C_VEL
LIN {X 0,Y 171.712,Z 522.621,A -85,B 0,C 180,E1 -24615.307,E2 -24615.307} C_VEL
LIN {X 0,Y 173.149,Z 509.444,A -85,B 0,C 180,E1 -24615.943,E2 -24615.943} C_VEL
LIN {X 0,Y 175.269,Z 476.762,A -85,B 0,C 180,E1 -24617.123,E2 -24617.123} C_VEL
LIN {X 0,Y 174.737,Z 474.36,A -85,B 0,C 180,E1 -24617.452,E2 -24617.452} C_VEL
LIN {X 0,Y 170.105,Z 461.96,A -85,B 0,C 180,E1 -24619.948,E2 -24619.948} C_VEL
LIN {X 0,Y 165.157,Z 451.095,A -85,B 0,C 180,E1 -24622.767,E2 -24622.767} C_VEL
LIN {X 0,Y 161.099,Z 443.286,A -85,B 0,C 180,E1 -24625.279,E2 -24625.279} C_VEL
LIN {X 0,Y 156.689,Z 435.435,A -85,B 0,C 180,E1 -24628.312,E2 -24628.312} C_VEL
LIN {X 0,Y 153.292,Z 430.685,A -85,B 0,C 180,E1 -24630.848,E2 -24630.848} C_VEL
LIN {X 0,Y 150.564,Z 427.053,A -85,B 0,C 180,E1 -24633.113,E2 -24633.113} C_VEL
LIN {X 0,Y 149.31,Z 425.734,A -85,B 0,C 180,E1 -24634.207,E2 -24634.207} C_VEL
LIN {X 0,Y 146.734,Z 422.533,A -85,B 0,C 180,E1 -24636.725,E2 -24636.725} C_VEL
LIN {X 0,Y 145.928,Z 421.084,A -85,B 0,C 180,E1 -24637.642,E2 -24637.642} C_VEL
LIN {X 0,Y 143.269,Z 418.891,A -85,B 0,C 180,E1 -24640.663,E2 -24640.663} C_VEL
LIN {X 0,Y 141.682,Z 415.824,A -85,B 0,C 180,E1 -24643.057,E2 -24643.057} C_VEL
LIN {X 0,Y 141.466,Z 415.477,A -85,B 0,C 180,E1 -24643.402,E2 -24643.402} C_VEL
LIN {X 0,Y 138.799,Z 413.92,A -85,B 0,C 180,E1 -24647.881,E2 -24647.881} C_VEL
LIN {X 0,Y 136.715,Z 410.231,A -85,B 0,C 180,E1 -24654.469,E2 -24654.469} C_VEL
LIN {X 0,Y 136.619,Z 409.445,A -85,B 0,C 180,E1 -24655.575,E2 -24655.575} C_VEL
LIN {X 0,Y 137.131,Z 409.396,A -85,B 0,C 180,E1 -24660,E2 -24660} C_VEL
LIN {X 0,Y 136.609,Z 409.54,A -85,B 0,C 180,E1 -24665.258,E2 -24665.258} C_VEL
LIN {X 0,Y 137.138,Z 411.426,A -85,B 0,C 180,E1 -24668.102,E2 -24668.102} C_VEL
LIN {X 0,Y 139.77,Z 414.754,A -85,B 0,C 180,E1 -24674.561,E2 -24674.561} C_VEL
LIN {X 0,Y 141.63,Z 415.624,A -85,B 0,C 180,E1 -24677.415,E2 -24677.415} C_VEL
LIN {X 0,Y 142.882,Z 418.359,A -85,B 0,C 180,E1 -24679.391,E2 -24679.391} C_VEL
LIN {X 0,Y 145.095,Z 420.641,A -85,B 0,C 180,E1 -24682.073,E2 -24682.073} C_VEL
LIN {X 0,Y 146.303,Z 421.621,A -85,B 0,C 180,E1 -24683.348,E2 -24683.348} C_VEL
LIN {X 0,Y 148.667,Z 425.148,A -85,B 0,C 180,E1 -24685.792,E2 -24685.792} C_VEL
LIN {X 0,Y 150.536,Z 426.971,A -85,B 0,C 180,E1 -24687.432,E2 -24687.432} C_VEL
LIN {X 0,Y 153.182,Z 430.612,A -85,B 0,C 180,E1 -24689.647,E2 -24689.647} C_VEL
LIN {X 0,Y 154.348,Z 432.114,A -85,B 0,C 180,E1 -24690.543,E2 -24690.543} C_VEL
LIN {X 0,Y 157.74,Z 436.825,A -85,B 0,C 180,E1 -24692.984,E2 -24692.984} C_VEL
LIN {X 0,Y 161.009,Z 441.578,A -85,B 0,C 180,E1 -24695.119,E2 -24695.119} C_VEL
LIN {X 0,Y 166.379,Z 450.035,A -85,B 0,C 180,E1 -24698.279,E2 -24698.279} C_VEL
LIN {X 0,Y 172.562,Z 461.111,A -85,B 0,C 180,E1 -24701.525,E2 -24701.525} C_VEL
LIN {X 0,Y 175.822,Z 467.868,A -85,B 0,C 180,E1 -24703.122,E2 -24703.122} C_VEL
LIN {X 0,Y 173.085,Z 507.041,A -85,B 0,C 180,E1 -24704.566,E2 -24704.566} C_VEL
LIN {X 0,Y 171.14,Z 520.654,A -85,B 0,C 180,E1 -24705.443,E2 -24705.443} C_VEL
LIN {X 0,Y 168.565,Z 533.455,A -85,B 0,C 180,E1 -24706.74,E2 -24706.74} C_VEL
LIN {X 0,Y 165.346,Z 545.227,A -85,B 0,C 180,E1 -24708.385,E2 -24708.385} C_VEL
LIN {X 0,Y 161.437,Z 556.545,A -85,B 0,C 180,E1 -24710.456,E2 -24710.456} C_VEL
LIN {X 0,Y 157.286,Z 566.742,A -85,B 0,C 180,E1 -24712.9,E2 -24712.9} C_VEL
LIN {X 0,Y 152.696,Z 576.807,A -85,B 0,C 180,E1 -24716.134,E2 -24716.134} C_VEL
LIN {X 0,Y 148.625,Z 584.771,A -85,B 0,C 180,E1 -24719.448,E2 -24719.448} C_VEL
LIN {X 0,Y 144.522,Z 591.925,A -85,B 0,C 180,E1 -24723.268,E2 -24723.268} C_VEL
LIN {X 0,Y 141.585,Z 596.745,A -85,B 0,C 180,E1 -24726.603,E2 -24726.603} C_VEL
LIN {X 0,Y 138.712,Z 601.424,A -85,B 0,C 180,E1 -24730.772,E2 -24730.772} C_VEL
LIN {X 0,Y 136.521,Z 605,A -85,B 0,C 180,E1 -24735.085,E2 -24735.085} C_VEL
LIN {X 0,Y 135.405,Z 606.845,A -85,B 0,C 180,E1 -24738.018,E2 -24738.018} C_VEL
LIN {X 0,Y 134.647,Z 608.227,A -85,B 0,C 180,E1 -24740.991,E2 -24740.991} C_VEL
LIN {X 0,Y 133.786,Z 609.814,A -85,B 0,C 180,E1 -24746.989,E2 -24746.989} C_VEL
LIN {X 0,Y 133.722,Z 610.039,A -85,B 0,C 180,E1 -24750,E2 -24750} C_VEL
LIN {X 0,Y 133.858,Z 609.69,A -85,B 0,C 180,E1 -24753.993,E2 -24753.993} C_VEL
LIN {X 0,Y 134.647,Z 608.295,A -85,B 0,C 180,E1 -24759.009,E2 -24759.009} C_VEL
LIN {X 0,Y 135.407,Z 606.943,A -85,B 0,C 180,E1 -24761.982,E2 -24761.982} C_VEL
LIN {X 0,Y 137.17,Z 604.079,A -85,B 0,C 180,E1 -24766.367,E2 -24766.367} C_VEL
LIN {X 0,Y 139.552,Z 600.195,A -85,B 0,C 180,E1 -24770.642,E2 -24770.642} C_VEL
LIN {X 0,Y 142.62,Z 595.18,A -85,B 0,C 180,E1 -24774.762,E2 -24774.762} C_VEL
LIN {X 0,Y 146.393,Z 588.856,A -85,B 0,C 180,E1 -24778.69,E2 -24778.69} C_VEL
LIN {X 0,Y 150.8,Z 580.941,A -85,B 0,C 180,E1 -24782.408,E2 -24782.408} C_VEL
LIN {X 0,Y 154.557,Z 573.057,A -85,B 0,C 180,E1 -24785.353,E2 -24785.353} C_VEL
LIN {X 0,Y 158.964,Z 563.033,A -85,B 0,C 180,E1 -24788.239,E2 -24788.239} C_VEL
LIN {X 0,Y 163.26,Z 551.929,A -85,B 0,C 180,E1 -24790.623,E2 -24790.623} C_VEL
LIN {X 0,Y 166.769,Z 541.042,A -85,B 0,C 180,E1 -24792.397,E2 -24792.397} C_VEL
LIN {X 0,Y 169.793,Z 529.004,A -85,B 0,C 180,E1 -24793.891,E2 -24793.891} C_VEL
LIN {X 0,Y 171.983,Z 517.25,A -85,B 0,C 180,E1 -24794.945,E2 -24794.945} C_VEL
LIN {X 0,Y 173.528,Z 504.504,A -85,B 0,C 180,E1 -24795.691,E2 -24795.691} C_VEL
LIN {X 0,Y 176.065,Z 468.149,A -85,B 0,C 180,E1 -24796.985,E2 -24796.985} C_VEL
LIN {X 0,Y 170.945,Z 457.995,A -85,B 0,C 180,E1 -24799.516,E2 -24799.516} C_VEL
LIN {X 0,Y 165.136,Z 447.929,A -85,B 0,C 180,E1 -24802.665,E2 -24802.665} C_VEL
LIN {X 0,Y 159.689,Z 439.397,A -85,B 0,C 180,E1 -24806.004,E2 -24806.004} C_VEL
LIN {X 0,Y 156.214,Z 434.676,A -85,B 0,C 180,E1 -24808.367,E2 -24808.367} C_VEL
LIN {X 0,Y 153.48,Z 430.871,A -85,B 0,C 180,E1 -24810.436,E2 -24810.436} C_VEL
LIN {X 0,Y 150.676,Z 427.157,A -85,B 0,C 180,E1 -24812.775,E2 -24812.775} C_VEL
LIN {X 0,Y 149.784,Z 426.112,A -85,B 0,C 180,E1 -24813.563,E2 -24813.563} C_VEL
LIN {X 0,Y 147.176,Z 423.211,A -85,B 0,C 180,E1 -24816.052,E2 -24816.052} C_VEL
LIN {X 0,Y 146.036,Z 421.111,A -85,B 0,C 180,E1 -24817.356,E2 -24817.356} C_VEL
LIN {X 0,Y 143.573,Z 419.236,A -85,B 0,C 180,E1 -24820.148,E2 -24820.148} C_VEL
LIN {X 0,Y 141.901,Z 416.347,A -85,B 0,C 180,E1 -24822.62,E2 -24822.62} C_VEL
LIN {X 0,Y 141.436,Z 415.453,A -85,B 0,C 180,E1 -24823.398,E2 -24823.398} C_VEL
LIN {X 0,Y 138.865,Z 413.947,A -85,B 0,C 180,E1 -24827.886,E2 -24827.886} C_VEL
LIN {X 0,Y 136.713,Z 409.988,A -85,B 0,C 180,E1 -24835.762,E2 -24835.762} C_VEL
LIN {X 0,Y 136.723,Z 409.436,A -85,B 0,C 180,E1 -24836.685,E2 -24836.685} C_VEL
LIN {X 0,Y 137.131,Z 409.393,A -85,B 0,C 180,E1 -24840,E2 -24840} C_VEL
LIN {X 0,Y 136.72,Z 409.599,A -85,B 0,C 180,E1 -24843.5,E2 -24843.5} C_VEL
LIN {X 0,Y 137.168,Z 411.58,A -85,B 0,C 180,E1 -24846.62,E2 -24846.62} C_VEL
LIN {X 0,Y 140.377,Z 415.063,A -85,B 0,C 180,E1 -24854.497,E2 -24854.497} C_VEL
LIN {X 0,Y 141.671,Z 415.701,A -85,B 0,C 180,E1 -24856.481,E2 -24856.481} C_VEL
LIN {X 0,Y 143.019,Z 418.523,A -85,B 0,C 180,E1 -24858.627,E2 -24858.627} C_VEL
LIN {X 0,Y 145.674,Z 420.973,A -85,B 0,C 180,E1 -24861.794,E2 -24861.794} C_VEL
LIN {X 0,Y 146.344,Z 421.655,A -85,B 0,C 180,E1 -24862.518,E2 -24862.518} C_VEL
LIN {X 0,Y 148.369,Z 424.809,A -85,B 0,C 180,E1 -24864.673,E2 -24864.673} C_VEL
LIN {X 0,Y 150.497,Z 426.903,A -85,B 0,C 180,E1 -24866.581,E2 -24866.581} C_VEL
LIN {X 0,Y 153.129,Z 430.509,A -85,B 0,C 180,E1 -24868.81,E2 -24868.81} C_VEL
LIN {X 0,Y 154.363,Z 432.124,A -85,B 0,C 180,E1 -24869.772,E2 -24869.772} C_VEL
LIN {X 0,Y 157.334,Z 436.492,A -85,B 0,C 180,E1 -24871.963,E2 -24871.963} C_VEL
LIN {X 0,Y 161.429,Z 443.706,A -85,B 0,C 180,E1 -24874.754,E2 -24874.754} C_VEL
LIN {X 0,Y 166.178,Z 453.034,A -85,B 0,C 180,E1 -24877.676,E2 -24877.676} C_VEL
LIN {X 0,Y 171.045,Z 464.062,A -85,B 0,C 180,E1 -24880.423,E2 -24880.423} C_VEL
LIN {X 0,Y 175.386,Z 476.03,A -85,B 0,C 180,E1 -24882.756,E2 -24882.756} C_VEL
LIN {X 0,Y 175.254,Z 481.005,A -85,B 0,C 180,E1 -24883.002,E2 -24883.002} C_VEL
LIN {X 0,Y 172.698,Z 516.559,A -85,B 0,C 180,E1 -24884.311,E2 -24884.311} C_VEL
LIN {X 0,Y 170.67,Z 529.88,A -85,B 0,C 180,E1 -24885.137,E2 -24885.137} C_VEL
LIN {X 0,Y 167.831,Z 542.417,A -85,B 0,C 180,E1 -24886.296,E2 -24886.296} C_VEL
LIN {X 0,Y 164.092,Z 555.077,A -85,B 0,C 180,E1 -24887.995,E2 -24887.995} C_VEL
LIN {X 0,Y 159.972,Z 566.342,A -85,B 0,C 180,E1 -24890.021,E2 -24890.021} C_VEL
LIN {X 0,Y 155.682,Z 576.494,A -85,B 0,C 180,E1 -24892.452,E2 -24892.452} C_VEL
LIN {X 0,Y 151.28,Z 585.647,A -85,B 0,C 180,E1 -24895.314,E2 -24895.314} C_VEL
LIN {X 0,Y 146.588,Z 594.576,A -85,B 0,C 180,E1 -24898.977,E2 -24898.977} C_VEL
LIN {X 0,Y 142.847,Z 601.636,A -85,B 0,C 180,E1 -24902.829,E2 -24902.829} C_VEL
LIN {X 0,Y 139.903,Z 606.631,A -85,B 0,C 180,E1 -24906.305,E2 -24906.305} C_VEL
LIN {X 0,Y 137.164,Z 611.358,A -85,B 0,C 180,E1 -24910.547,E2 -24910.547} C_VEL
LIN {X 0,Y 135.233,Z 614.978,A -85,B 0,C 180,E1 -24914.939,E2 -24914.939} C_VEL
LIN {X 0,Y 134.378,Z 616.849,A -85,B 0,C 180,E1 -24917.925,E2 -24917.925} C_VEL
LIN {X 0,Y 133.817,Z 618.255,A -85,B 0,C 180,E1 -24920.935,E2 -24920.935} C_VEL
LIN {X 0,Y 133.539,Z 619.263,A -85,B 0,C 180,E1 -24923.958,E2 -24923.958} C_VEL
LIN {X 0,Y 133.542,Z 620.068,A -85,B 0,C 180,E1 -24929.291,E2 -24929.291} C_VEL
LIN {X 0,Y 133.485,Z 619.865,A -85,B 0,C 180,E1 -24933.018,E2 -24933.018} C_VEL
LIN {X 0,Y 133.54,Z 619.238,A -85,B 0,C 180,E1 -24936.042,E2 -24936.042} C_VEL
LIN {X 0,Y 133.811,Z 618.22,A -85,B 0,C 180,E1 -24939.065,E2 -24939.065} C_VEL
LIN {X 0,Y 134.461,Z 616.536,A -85,B 0,C 180,E1 -24942.493,E2 -24942.493} C_VEL
LIN {X 0,Y 134.492,Z 615.039,A -85,B 0,C 180,E1 -24944.922,E2 -24944.922} C_VEL
LIN {X 0,Y 133.233,Z 612.057,A -85,B 0,C 180,E1 -24948.951,E2 -24948.951} C_VEL
LIN {X 0,Y 132.614,Z 608.477,A -85,B 0,C 180,E1 -24952.932,E2 -24952.932} C_VEL
LIN {X 0,Y 133.613,Z 605.911,A -85,B 0,C 180,E1 -24955.182,E2 -24955.182} C_VEL
LIN {X 0,Y 137.152,Z 600.13,A -85,B 0,C 180,E1 -24959.209,E2 -24959.209} C_VEL
LIN {X 0,Y 141.32,Z 592.76,A -85,B 0,C 180,E1 -24963.163,E2 -24963.163} C_VEL
LIN {X 0,Y 145.493,Z 585.154,A -85,B 0,C 180,E1 -24966.279,E2 -24966.279} C_VEL
LIN {X 0,Y 150.131,Z 575.95,A -85,B 0,C 180,E1 -24969.194,E2 -24969.194} C_VEL
LIN {X 0,Y 154.589,Z 565.713,A -85,B 0,C 180,E1 -24971.673,E2 -24971.673} C_VEL
LIN {X 0,Y 158.877,Z 554.368,A -85,B 0,C 180,E1 -24973.722,E2 -24973.722} C_VEL
LIN {X 0,Y 162.489,Z 542.586,A -85,B 0,C 180,E1 -24975.312,E2 -24975.312} C_VEL
LIN {X 0,Y 165.478,Z 529.886,A -85,B 0,C 180,E1 -24976.515,E2 -24976.515} C_VEL
LIN {X 0,Y 167.607,Z 516.13,A -85,B 0,C 180,E1 -24977.391,E2 -24977.391} C_VEL
LIN {X 0,Y 170.403,Z 478.201,A -85,B 0,C 180,E1 -24978.808,E2 -24978.808} C_VEL
LIN {X 0,Y 166.167,Z 466.442,A -85,B 0,C 180,E1 -24981.272,E2 -24981.272} C_VEL
LIN {X 0,Y 161.535,Z 455.777,A -85,B 0,C 180,E1 -24984.127,E2 -24984.127} C_VEL
LIN {X 0,Y 156.47,Z 445.711,A -85,B 0,C 180,E1 -24987.576,E2 -24987.576} C_VEL
LIN {X 0,Y 153.26,Z 440.205,A -85,B 0,C 180,E1 -24989.992,E2 -24989.992} C_VEL
LIN {X 0,Y 150.929,Z 436.846,A -85,B 0,C 180,E1 -24991.87,E2 -24991.87} C_VEL
LIN {X 0,Y 147.8,Z 432.611,A -85,B 0,C 180,E1 -24994.662,E2 -24994.662} C_VEL
LIN {X 0,Y 144.946,Z 429.137,A -85,B 0,C 180,E1 -24997.558,E2 -24997.558} C_VEL
LIN {X 0,Y 144.154,Z 427.751,A -85,B 0,C 180,E1 -24998.503,E2 -24998.503} C_VEL
LIN {X 0,Y 141.403,Z 425.096,A -85,B 0,C 180,E1 -25001.902,E2 -25001.902} C_VEL
LIN {X 0,Y 139.912,Z 422.328,A -85,B 0,C 180,E1 -25004.336,E2 -25004.336} C_VEL
LIN {X 0,Y 137.424,Z 420.502,A -85,B 0,C 180,E1 -25008.965,E2 -25008.965} C_VEL
LIN {X 0,Y 135.69,Z 416.931,A -85,B 0,C 180,E1 -25015.358,E2 -25015.358} C_VEL
LIN {X 0,Y 135.578,Z 416.45,A -85,B 0,C 180,E1 -25016.285,E2 -25016.285} C_VEL
LIN {X 0,Y 135.402,Z 416.402,A -85,B 0,C 180,E1 -25022.975,E2 -25022.975} C_VEL
LIN {X 0,Y 135.647,Z 416.666,A -85,B 0,C 180,E1 -25024.83,E2 -25024.83} C_VEL
LIN {X 0,Y 137.814,Z 421.018,A -85,B 0,C 180,E1 -25032.517,E2 -25032.517} C_VEL
LIN {X 0,Y 140.179,Z 422.589,A -85,B 0,C 180,E1 -25036.662,E2 -25036.662} C_VEL
LIN {X 0,Y 141.822,Z 425.649,A -85,B 0,C 180,E1 -25039.26,E2 -25039.26} C_VEL
LIN {X 0,Y 144.473,Z 428.205,A -85,B 0,C 180,E1 -25042.445,E2 -25042.445} C_VEL
LIN {X 0,Y 146.943,Z 431.827,A -85,B 0,C 180,E1 -25045.118,E2 -25045.118} C_VEL
LIN {X 0,Y 148.4,Z 433.366,A -85,B 0,C 180,E1 -25046.472,E2 -25046.472} C_VEL
LIN {X 0,Y 151.298,Z 437.26,A -85,B 0,C 180,E1 -25049.002,E2 -25049.002} C_VEL
LIN {X 0,Y 155.528,Z 443.439,A -85,B 0,C 180,E1 -25052.261,E2 -25052.261} C_VEL
LIN {X 0,Y 159.394,Z 449.255,A -85,B 0,C 180,E1 -25054.877,E2 -25054.877} C_VEL
LIN {X 0,Y 165.065,Z 459.032,A -85,B 0,C 180,E1 -25058.318,E2 -25058.318} C_VEL
LIN {X 0,Y 170.378,Z 469.331,A -85,B 0,C 180,E1 -25061.201,E2 -25061.201} C_VEL
LIN {X 0,Y 170.895,Z 470.481,A -85,B 0,C 180,E1 -25061.473,E2 -25061.473} C_VEL
LIN {X 0,Y 168.182,Z 507.432,A -85,B 0,C 180,E1 -25062.854,E2 -25062.854} C_VEL
LIN {X 0,Y 166.135,Z 521.13,A -85,B 0,C 180,E1 -25063.747,E2 -25063.747} C_VEL
LIN {X 0,Y 163.472,Z 533.728,A -85,B 0,C 180,E1 -25065.036,E2 -25065.036} C_VEL
LIN {X 0,Y 160.125,Z 545.498,A -85,B 0,C 180,E1 -25066.703,E2 -25066.703} C_VEL
LIN {X 0,Y 156.045,Z 556.816,A -85,B 0,C 180,E1 -25068.802,E2 -25068.802} C_VEL
LIN {X 0,Y 151.692,Z 567.012,A -85,B 0,C 180,E1 -25071.285,E2 -25071.285} C_VEL
LIN {X 0,Y 147.344,Z 576.153,A -85,B 0,C 180,E1 -25074.247,E2 -25074.247} C_VEL
LIN {X 0,Y 142.562,Z 585.04,A -85,B 0,C 180,E1 -25077.999,E2 -25077.999} C_VEL
LIN {X 0,Y 138.212,Z 592.195,A -85,B 0,C 180,E1 -25081.943,E2 -25081.943} C_VEL
LIN {X 0,Y 135.088,Z 597.014,A -85,B 0,C 180,E1 -25085.405,E2 -25085.405} C_VEL
LIN {X 0,Y 132.033,Z 601.693,A -85,B 0,C 180,E1 -25089.758,E2 -25089.758} C_VEL
LIN {X 0,Y 129.665,Z 605.268,A -85,B 0,C 180,E1 -25094.276,E2 -25094.276} C_VEL
LIN {X 0,Y 128.474,Z 607.113,A -85,B 0,C 180,E1 -25097.361,E2 -25097.361} C_VEL
LIN {X 0,Y 127.634,Z 608.495,A -85,B 0,C 180,E1 -25100.492,E2 -25100.492} C_VEL
LIN {X 0,Y 126.7,Z 610.082,A -85,B 0,C 180,E1 -25106.82,E2 -25106.82} C_VEL
LIN {X 0,Y 126.633,Z 610.305,A -85,B 0,C 180,E1 -25110,E2 -25110} C_VEL
LIN {X 0,Y 126.7,Z 610.111,A -85,B 0,C 180,E1 -25113.18,E2 -25113.18} C_VEL
LIN {X 0,Y 127.634,Z 608.562,A -85,B 0,C 180,E1 -25119.508,E2 -25119.508} C_VEL
LIN {X 0,Y 128.476,Z 607.209,A -85,B 0,C 180,E1 -25122.639,E2 -25122.639} C_VEL
LIN {X 0,Y 130.366,Z 604.346,A -85,B 0,C 180,E1 -25127.247,E2 -25127.247} C_VEL
LIN {X 0,Y 132.939,Z 600.461,A -85,B 0,C 180,E1 -25131.719,E2 -25131.719} C_VEL
LIN {X 0,Y 136.207,Z 595.446,A -85,B 0,C 180,E1 -25136.013,E2 -25136.013} C_VEL
LIN {X 0,Y 140.216,Z 589.121,A -85,B 0,C 180,E1 -25140.08,E2 -25140.08} C_VEL
LIN {X 0,Y 144.839,Z 581.23,A -85,B 0,C 180,E1 -25143.904,E2 -25143.904} C_VEL
LIN {X 0,Y 148.894,Z 573.147,A -85,B 0,C 180,E1 -25146.998,E2 -25146.998} C_VEL
LIN {X 0,Y 153.463,Z 563.296,A -85,B 0,C 180,E1 -25149.876,E2 -25149.876} C_VEL
LIN {X 0,Y 157.956,Z 552.191,A -85,B 0,C 180,E1 -25152.295,E2 -25152.295} C_VEL
LIN {X 0,Y 161.615,Z 541.302,A -85,B 0,C 180,E1 -25154.088,E2 -25154.088} C_VEL
LIN {X 0,Y 164.757,Z 529.264,A -85,B 0,C 180,E1 -25155.601,E2 -25155.601} C_VEL
LIN {X 0,Y 167.069,Z 517.398,A -85,B 0,C 180,E1 -25156.668,E2 -25156.668} C_VEL
LIN {X 0,Y 168.709,Z 504.097,A -85,B 0,C 180,E1 -25157.442,E2 -25157.442} C_VEL
LIN {X 0,Y 171.123,Z 470.748,A -85,B 0,C 180,E1 -25158.642,E2 -25158.642} C_VEL
LIN {X 0,Y 165.881,Z 460.337,A -85,B 0,C 180,E1 -25161.469,E2 -25161.469} C_VEL
LIN {X 0,Y 160.509,Z 451.051,A -85,B 0,C 180,E1 -25164.67,E2 -25164.67} C_VEL
LIN {X 0,Y 155.979,Z 444.001,A -85,B 0,C 180,E1 -25167.707,E2 -25167.707} C_VEL
LIN {X 0,Y 153.368,Z 440.274,A -85,B 0,C 180,E1 -25169.64,E2 -25169.64} C_VEL
LIN {X 0,Y 150.846,Z 436.736,A -85,B 0,C 180,E1 -25171.684,E2 -25171.684} C_VEL
LIN {X 0,Y 147.843,Z 432.64,A -85,B 0,C 180,E1 -25174.402,E2 -25174.402} C_VEL
LIN {X 0,Y 145.037,Z 429.214,A -85,B 0,C 180,E1 -25177.282,E2 -25177.282} C_VEL
LIN {X 0,Y 144.213,Z 427.77,A -85,B 0,C 180,E1 -25178.279,E2 -25178.279} C_VEL
LIN {X 0,Y 141.586,Z 425.319,A -85,B 0,C 180,E1 -25181.552,E2 -25181.552} C_VEL
LIN {X 0,Y 140.132,Z 422.396,A -85,B 0,C 180,E1 -25183.988,E2 -25183.988} C_VEL
LIN {X 0,Y 137.633,Z 420.729,A -85,B 0,C 180,E1 -25188.666,E2 -25188.666} C_VEL
LIN {X 0,Y 135.756,Z 416.69,A -85,B 0,C 180,E1 -25196.661,E2 -25196.661} C_VEL
LIN {X 0,Y 135.604,Z 416.327,A -85,B 0,C 180,E1 -25200,E2 -25200} C_VEL
LIN {X 0,Y 135.775,Z 416.66,A -85,B 0,C 180,E1 -25202.967,E2 -25202.967} C_VEL
LIN {X 0,Y 136.475,Z 419.087,A -85,B 0,C 180,E1 -25207.397,E2 -25207.397} C_VEL
LIN {X 0,Y 139.324,Z 422.054,A -85,B 0,C 180,E1 -25214.236,E2 -25214.236} C_VEL
LIN {X 0,Y 140.231,Z 422.672,A -85,B 0,C 180,E1 -25215.721,E2 -25215.721} C_VEL
LIN {X 0,Y 142.149,Z 426.002,A -85,B 0,C 180,E1 -25218.746,E2 -25218.746} C_VEL
LIN {X 0,Y 144.484,Z 428.168,A -85,B 0,C 180,E1 -25221.561,E2 -25221.561} C_VEL
LIN {X 0,Y 146.704,Z 431.522,A -85,B 0,C 180,E1 -25224.029,E2 -25224.029} C_VEL
LIN {X 0,Y 148.41,Z 433.319,A -85,B 0,C 180,E1 -25225.647,E2 -25225.647} C_VEL
LIN {X 0,Y 152.064,Z 438.425,A -85,B 0,C 180,E1 -25228.842,E2 -25228.842} C_VEL
LIN {X 0,Y 154.474,Z 442.071,A -85,B 0,C 180,E1 -25230.735,E2 -25230.735} C_VEL
LIN {X 0,Y 158.743,Z 449.877,A -85,B 0,C 180,E1 -25233.835,E2 -25233.835} C_VEL
LIN {X 0,Y 163.776,Z 460.557,A -85,B 0,C 180,E1 -25237.12,E2 -25237.12} C_VEL
LIN {X 0,Y 167.881,Z 470.549,A -85,B 0,C 180,E1 -25239.576,E2 -25239.576} C_VEL
LIN {X 0,Y 170.579,Z 478.376,A -85,B 0,C 180,E1 -25241.142,E2 -25241.142} C_VEL
LIN {X 0,Y 167.787,Z 516.519,A -85,B 0,C 180,E1 -25242.586,E2 -25242.586} C_VEL
LIN {X 0,Y 165.664,Z 529.895,A -85,B 0,C 180,E1 -25243.427,E2 -25243.427} C_VEL
LIN {X 0,Y 162.774,Z 542.156,A -85,B 0,C 180,E1 -25244.57,E2 -25244.57} C_VEL
LIN {X 0,Y 158.893,Z 554.815,A -85,B 0,C 180,E1 -25246.283,E2 -25246.283} C_VEL
LIN {X 0,Y 154.604,Z 566.079,A -85,B 0,C 180,E1 -25248.333,E2 -25248.333} C_VEL
LIN {X 0,Y 150.123,Z 576.23,A -85,B 0,C 180,E1 -25250.803,E2 -25250.803} C_VEL
LIN {X 0,Y 145.472,Z 585.381,A -85,B 0,C 180,E1 -25253.715,E2 -25253.715} C_VEL
LIN {X 0,Y 140.522,Z 594.31,A -85,B 0,C 180,E1 -25257.477,E2 -25257.477} C_VEL
LIN {X 0,Y 136.831,Z 600.705,A -85,B 0,C 180,E1 -25261.034,E2 -25261.034} C_VEL
LIN {X 0,Y 133.402,Z 606.364,A -85,B 0,C 180,E1 -25265.074,E2 -25265.074} C_VEL
LIN {X 0,Y 130.471,Z 611.091,A -85,B 0,C 180,E1 -25269.505,E2 -25269.505} C_VEL
LIN {X 0,Y 128.356,Z 614.711,A -85,B 0,C 180,E1 -25274.112,E2 -25274.112} C_VEL
LIN {X 0,Y 127.409,Z 616.581,A -85,B 0,C 180,E1 -25277.253,E2 -25277.253} C_VEL
LIN {X 0,Y 126.782,Z 617.987,A -85,B 0,C 180,E1 -25280.427,E2 -25280.427} C_VEL
LIN {X 0,Y 126.46,Z 618.995,A -85,B 0,C 180,E1 -25283.619,E2 -25283.619} C_VEL
LIN {X 0,Y 126.378,Z 619.613,A -85,B 0,C 180,E1 -25286.812,E2 -25286.812} C_VEL
LIN {X 0,Y 126.507,Z 619.818,A -85,B 0,C 180,E1 -25290.357,E2 -25290.357} C_VEL
LIN {X 0,Y 126.46,Z 618.97,A -85,B 0,C 180,E1 -25296.381,E2 -25296.381} C_VEL
LIN {X 0,Y 126.776,Z 617.951,A -85,B 0,C 180,E1 -25299.573,E2 -25299.573} C_VEL
LIN {X 0,Y 127.413,Z 616.487,A -85,B 0,C 180,E1 -25302.818,E2 -25302.818} C_VEL
LIN {X 0,Y 128.925,Z 613.557,A -85,B 0,C 180,E1 -25307.446,E2 -25307.446} C_VEL
LIN {X 0,Y 131.383,Z 609.553,A -85,B 0,C 180,E1 -25311.99,E2 -25311.99} C_VEL
LIN {X 0,Y 133.613,Z 605.911,A -85,B 0,C 180,E1 -25315.182,E2 -25315.182} C_VEL
LIN {X 0,Y 134.756,Z 603.152,A -85,B 0,C 180,E1 -25317.353,E2 -25317.353} C_VEL
LIN {X 0,Y 135.127,Z 598.255,A -85,B 0,C 180,E1 -25321.017,E2 -25321.017} C_VEL
LIN {X 0,Y 135.822,Z 592.799,A -85,B 0,C 180,E1 -25324.516,E2 -25324.516} C_VEL
LIN {X 0,Y 137.405,Z 589.092,A -85,B 0,C 180,E1 -25326.342,E2 -25326.342} C_VEL
LIN {X 0,Y 142.677,Z 579.596,A -85,B 0,C 180,E1 -25329.817,E2 -25329.817} C_VEL
LIN {X 0,Y 147.778,Z 569.077,A -85,B 0,C 180,E1 -25332.663,E2 -25332.663} C_VEL
LIN {X 0,Y 152.667,Z 557.237,A -85,B 0,C 180,E1 -25335.054,E2 -25335.054} C_VEL
LIN {X 0,Y 156.691,Z 545.3,A -85,B 0,C 180,E1 -25336.789,E2 -25336.789} C_VEL
LIN {X 0,Y 159.961,Z 532.872,A -85,B 0,C 180,E1 -25338.086,E2 -25338.086} C_VEL
LIN {X 0,Y 162.332,Z 520.241,A -85,B 0,C 180,E1 -25338.993,E2 -25338.993} C_VEL
LIN {X 0,Y 163.86,Z 505.306,A -85,B 0,C 180,E1 -25339.646,E2 -25339.646} C_VEL
LIN {X 0,Y 165.613,Z 480.367,A -85,B 0,C 180,E1 -25340.575,E2 -25340.575} C_VEL
LIN {X 0,Y 162.081,Z 470.249,A -85,B 0,C 180,E1 -25342.818,E2 -25342.818} C_VEL
LIN {X 0,Y 158.003,Z 460.504,A -85,B 0,C 180,E1 -25345.547,E2 -25345.547} C_VEL
LIN {X 0,Y 153.366,Z 450.899,A -85,B 0,C 180,E1 -25348.967,E2 -25348.967} C_VEL
LIN {X 0,Y 150.596,Z 445.993,A -85,B 0,C 180,E1 -25351.213,E2 -25351.213} C_VEL
LIN {X 0,Y 148.348,Z 442.68,A -85,B 0,C 180,E1 -25353.157,E2 -25353.157} C_VEL
LIN {X 0,Y 145.615,Z 438.852,A -85,B 0,C 180,E1 -25355.78,E2 -25355.78} C_VEL
LIN {X 0,Y 142.776,Z 434.98,A -85,B 0,C 180,E1 -25358.931,E2 -25358.931} C_VEL
LIN {X 0,Y 141.42,Z 433.568,A -85,B 0,C 180,E1 -25360.59,E2 -25360.59} C_VEL
LIN {X 0,Y 139.198,Z 430.45,A -85,B 0,C 180,E1 -25363.878,E2 -25363.878} C_VEL
LIN {X 0,Y 138.567,Z 429.203,A -85,B 0,C 180,E1 -25365.028,E2 -25365.028} C_VEL
LIN {X 0,Y 136.017,Z 427.011,A -85,B 0,C 180,E1 -25370.287,E2 -25370.287} C_VEL
LIN {X 0,Y 134.701,Z 423.603,A -85,B 0,C 180,E1 -25376.261,E2 -25376.261} C_VEL
LIN {X 0,Y 134.408,Z 423.298,A -85,B 0,C 180,E1 -25380,E2 -25380} C_VEL
LIN {X 0,Y 134.694,Z 423.649,A -85,B 0,C 180,E1 -25384.302,E2 -25384.302} C_VEL
LIN {X 0,Y 136.818,Z 428.051,A -85,B 0,C 180,E1 -25392.298,E2 -25392.298} C_VEL
LIN {X 0,Y 138.799,Z 429.562,A -85,B 0,C 180,E1 -25395.962,E2 -25395.962} C_VEL
LIN {X 0,Y 140.648,Z 432.721,A -85,B 0,C 180,E1 -25398.954,E2 -25398.954} C_VEL
LIN {X 0,Y 142.795,Z 434.969,A -85,B 0,C 180,E1 -25401.662,E2 -25401.662} C_VEL
LIN {X 0,Y 145.283,Z 438.545,A -85,B 0,C 180,E1 -25404.47,E2 -25404.47} C_VEL
LIN {X 0,Y 146.583,Z 440.152,A -85,B 0,C 180,E1 -25405.757,E2 -25405.757} C_VEL
LIN {X 0,Y 149.762,Z 444.71,A -85,B 0,C 180,E1 -25408.656,E2 -25408.656} C_VEL
LIN {X 0,Y 152.653,Z 449.001,A -85,B 0,C 180,E1 -25410.994,E2 -25410.994} C_VEL
LIN {X 0,Y 156.372,Z 454.83,A -85,B 0,C 180,E1 -25413.696,E2 -25413.696} C_VEL
LIN {X 0,Y 161.614,Z 464.155,A -85,B 0,C 180,E1 -25417.099,E2 -25417.099} C_VEL
LIN {X 0,Y 166.136,Z 473.177,A -85,B 0,C 180,E1 -25419.74,E2 -25419.74} C_VEL
LIN {X 0,Y 163.443,Z 507.718,A -85,B 0,C 180,E1 -25421.033,E2 -25421.033} C_VEL
LIN {X 0,Y 161.39,Z 521.052,A -85,B 0,C 180,E1 -25421.903,E2 -25421.903} C_VEL
LIN {X 0,Y 158.546,Z 534.001,A -85,B 0,C 180,E1 -25423.229,E2 -25423.229} C_VEL
LIN {X 0,Y 155.042,Z 545.77,A -85,B 0,C 180,E1 -25424.907,E2 -25424.907} C_VEL
LIN {X 0,Y 150.775,Z 557.087,A -85,B 0,C 180,E1 -25427.024,E2 -25427.024} C_VEL
LIN {X 0,Y 146.223,Z 567.282,A -85,B 0,C 180,E1 -25429.546,E2 -25429.546} C_VEL
LIN {X 0,Y 141.831,Z 576.105,A -85,B 0,C 180,E1 -25432.451,E2 -25432.451} C_VEL
LIN {X 0,Y 137.395,Z 583.964,A -85,B 0,C 180,E1 -25435.76,E2 -25435.76} C_VEL
LIN {X 0,Y 132.734,Z 591.354,A -85,B 0,C 180,E1 -25439.802,E2 -25439.802} C_VEL
LIN {X 0,Y 128.657,Z 597.284,A -85,B 0,C 180,E1 -25444.088,E2 -25444.088} C_VEL
LIN {X 0,Y 125.405,Z 601.961,A -85,B 0,C 180,E1 -25448.638,E2 -25448.638} C_VEL
LIN {X 0,Y 122.848,Z 605.536,A -85,B 0,C 180,E1 -25453.379,E2 -25453.379} C_VEL
LIN {X 0,Y 121.573,Z 607.38,A -85,B 0,C 180,E1 -25456.631,E2 -25456.631} C_VEL
LIN {X 0,Y 120.627,Z 608.763,A -85,B 0,C 180,E1 -25459.934,E2 -25459.934} C_VEL
LIN {X 0,Y 119.625,Z 610.349,A -85,B 0,C 180,E1 -25466.632,E2 -25466.632} C_VEL
LIN {X 0,Y 119.528,Z 610.507,A -85,B 0,C 180,E1 -25471.683,E2 -25471.683} C_VEL
LIN {X 0,Y 119.987,Z 609.793,A -85,B 0,C 180,E1 -25476.727,E2 -25476.727} C_VEL
LIN {X 0,Y 121.574,Z 607.475,A -85,B 0,C 180,E1 -25483.369,E2 -25483.369} C_VEL
LIN {X 0,Y 123.604,Z 604.612,A -85,B 0,C 180,E1 -25488.223,E2 -25488.223} C_VEL
LIN {X 0,Y 126.382,Z 600.727,A -85,B 0,C 180,E1 -25492.908,E2 -25492.908} C_VEL
LIN {X 0,Y 129.87,Z 595.711,A -85,B 0,C 180,E1 -25497.385,E2 -25497.385} C_VEL
LIN {X 0,Y 134.134,Z 589.385,A -85,B 0,C 180,E1 -25501.597,E2 -25501.597} C_VEL
LIN {X 0,Y 138.865,Z 581.719,A -85,B 0,C 180,E1 -25505.442,E2 -25505.442} C_VEL
LIN {X 0,Y 143.192,Z 573.587,A -85,B 0,C 180,E1 -25508.648,E2 -25508.648} C_VEL
LIN {X 0,Y 148.085,Z 563.559,A -85,B 0,C 180,E1 -25511.637,E2 -25511.637} C_VEL
LIN {X 0,Y 152.792,Z 552.453,A -85,B 0,C 180,E1 -25514.082,E2 -25514.082} C_VEL
LIN {X 0,Y 156.602,Z 541.563,A -85,B 0,C 180,E1 -25515.892,E2 -25515.892} C_VEL
LIN {X 0,Y 159.869,Z 529.523,A -85,B 0,C 180,E1 -25517.419,E2 -25517.419} C_VEL
LIN {X 0,Y 162.394,Z 516.971,A -85,B 0,C 180,E1 -25518.538,E2 -25518.538} C_VEL
LIN {X 0,Y 164.022,Z 503.995,A -85,B 0,C 180,E1 -25519.284,E2 -25519.284} C_VEL
LIN {X 0,Y 166.347,Z 473.424,A -85,B 0,C 180,E1 -25520.385,E2 -25520.385} C_VEL
LIN {X 0,Y 161.055,Z 462.979,A -85,B 0,C 180,E1 -25523.504,E2 -25523.504} C_VEL
LIN {X 0,Y 156.281,Z 454.505,A -85,B 0,C 180,E1 -25526.655,E2 -25526.655} C_VEL
LIN {X 0,Y 151.439,Z 447.038,A -85,B 0,C 180,E1 -25530.278,E2 -25530.278} C_VEL
LIN {X 0,Y 148.483,Z 442.803,A -85,B 0,C 180,E1 -25532.803,E2 -25532.803} C_VEL
LIN {X 0,Y 145.768,Z 438.974,A -85,B 0,C 180,E1 -25535.427,E2 -25535.427} C_VEL
LIN {X 0,Y 143.047,Z 435.369,A -85,B 0,C 180,E1 -25538.446,E2 -25538.446} C_VEL
LIN {X 0,Y 142.327,Z 434.313,A -85,B 0,C 180,E1 -25539.351,E2 -25539.351} C_VEL
LIN {X 0,Y 139.74,Z 431.378,A -85,B 0,C 180,E1 -25542.928,E2 -25542.928} C_VEL
LIN {X 0,Y 138.629,Z 429.226,A -85,B 0,C 180,E1 -25544.94,E2 -25544.94} C_VEL
LIN {X 0,Y 135.877,Z 426.778,A -85,B 0,C 180,E1 -25551.073,E2 -25551.073} C_VEL
LIN {X 0,Y 134.807,Z 423.475,A -85,B 0,C 180,E1 -25557.759,E2 -25557.759} C_VEL
LIN {X 0,Y 134.855,Z 423.608,A -85,B 0,C 180,E1 -25562.427,E2 -25562.427} C_VEL
LIN {X 0,Y 135.913,Z 426.806,A -85,B 0,C 180,E1 -25568.549,E2 -25568.549} C_VEL
LIN {X 0,Y 138.832,Z 429.507,A -85,B 0,C 180,E1 -25574.943,E2 -25574.943} C_VEL
LIN {X 0,Y 140.881,Z 432.955,A -85,B 0,C 180,E1 -25578.308,E2 -25578.308} C_VEL
LIN {X 0,Y 142.746,Z 434.832,A -85,B 0,C 180,E1 -25580.684,E2 -25580.684} C_VEL
LIN {X 0,Y 145.216,Z 438.405,A -85,B 0,C 180,E1 -25583.533,E2 -25583.533} C_VEL
LIN {X 0,Y 146.496,Z 439.94,A -85,B 0,C 180,E1 -25584.82,E2 -25584.82} C_VEL
LIN {X 0,Y 149.809,Z 444.731,A -85,B 0,C 180,E1 -25587.886,E2 -25587.886} C_VEL
